LIN {X 0,Y 580.276,Z 358.823,A -85,B 0,C 180,E1 -1965.982,E2 -1965.982} C_VEL
LIN {X 0,Y 580.288,Z 358.825,A -85,B 0,C 180,E1 -1968.827,E2 -1968.827} C_VEL
LIN {X 0,Y 580.269,Z 358.822,A -85,B 0,C 180,E1 -1971.643,E2 -1971.643} C_VEL
LIN {X 0,Y 580.294,Z 358.829,A -85,B 0,C 180,E1 -1974.44,E2 -1974.44} C_VEL
LIN {X 0,Y 580.294,Z 358.821,A -85,B 0,C 180,E1 -1977.223,E2 -1977.223} C_VEL
LIN {X 0,Y 580.311,Z 358.82,A -85,B 0,C 180,E1 -1980,E2 -1980} C_VEL
LIN {X 0,Y 580.319,Z 358.824,A -85,B 0,C 180,E1 -1982.777,E2 -1982.777} C_VEL
LIN {X 0,Y 580.273,Z 358.822,A -85,B 0,C 180,E1 -1985.56,E2 -1985.56} C_VEL
LIN {X 0,Y 580.238,Z 358.826,A -85,B 0,C 180,E1 -1987.657,E2 -1987.657} C_VEL
LIN {X 0,Y 580.25,Z 358.833,A -85,B 0,C 180,E1 -1990.468,E2 -1990.468} C_VEL
LIN {X 0,Y 580.275,Z 358.83,A -85,B 0,C 180,E1 -1992.592,E2 -1992.592} C_VEL
LIN {X 0,Y 580.261,Z 358.824,A -85,B 0,C 180,E1 -1995.454,E2 -1995.454} C_VEL
LIN {X 0,Y 580.245,Z 358.825,A -85,B 0,C 180,E1 -1997.626,E2 -1997.626} C_VEL
LIN {X 0,Y 580.26,Z 358.824,A -85,B 0,C 180,E1 -1999.824,E2 -1999.824} C_VEL
LIN {X 0,Y 580.262,Z 358.824,A -85,B 0,C 180,E1 -2001.343,E2 -2001.343} C_VEL
LIN {X 0,Y 579.556,Z 358.913,A -85,B 0,C 180,E1 -2001.923,E2 -2001.923} C_VEL
LIN {X 0,Y 576.673,Z 359.279,A -85,B 0,C 180,E1 -2002.862,E2 -2002.862} C_VEL
LIN {X 0,Y 574.271,Z 359.574,A -85,B 0,C 180,E1 -2003.618,E2 -2003.618} C_VEL
LIN {X 0,Y 573.259,Z 359.7,A -85,B 0,C 180,E1 -2004.202,E2 -2004.202} C_VEL
LIN {X 0,Y 573.185,Z 359.711,A -85,B 0,C 180,E1 -2004.4,E2 -2004.4} C_VEL
LIN {X 0,Y 573.168,Z 359.714,A -85,B 0,C 180,E1 -2006.98,E2 -2006.98} C_VEL
LIN {X 0,Y 573.197,Z 359.704,A -85,B 0,C 180,E1 -2009.483,E2 -2009.483} C_VEL
LIN {X 0,Y 573.224,Z 359.704,A -85,B 0,C 180,E1 -2012.227,E2 -2012.227} C_VEL
LIN {X 0,Y 573.213,Z 359.712,A -85,B 0,C 180,E1 -2014.771,E2 -2014.771} C_VEL
LIN {X 0,Y 573.201,Z 359.7,A -85,B 0,C 180,E1 -2017.81,E2 -2017.81} C_VEL
LIN {X 0,Y 573.233,Z 359.706,A -85,B 0,C 180,E1 -2020.526,E2 -2020.526} C_VEL
LIN {X 0,Y 573.191,Z 359.705,A -85,B 0,C 180,E1 -2023.666,E2 -2023.666} C_VEL
LIN {X 0,Y 573.184,Z 359.713,A -85,B 0,C 180,E1 -2026.638,E2 -2026.638} C_VEL
LIN {X 0,Y 573.218,Z 359.702,A -85,B 0,C 180,E1 -2029.478,E2 -2029.478} C_VEL
LIN {X 0,Y 573.21,Z 359.705,A -85,B 0,C 180,E1 -2032.192,E2 -2032.192} C_VEL
LIN {X 0,Y 573.205,Z 359.703,A -85,B 0,C 180,E1 -2035.233,E2 -2035.233} C_VEL
LIN {X 0,Y 573.226,Z 359.706,A -85,B 0,C 180,E1 -2037.776,E2 -2037.776} C_VEL
LIN {X 0,Y 573.237,Z 359.888,A -85,B 0,C 180,E1 -2039.418,E2 -2039.418} C_VEL
LIN {X 0,Y 575.578,Z 368.52,A -85,B 0,C 180,E1 -2040.393,E2 -2040.393} C_VEL
LIN {X 0,Y 575.413,Z 394.138,A -85,B 0,C 180,E1 -2042.851,E2 -2042.851} C_VEL
LIN {X 0,Y 574.972,Z 420.796,A -85,B 0,C 180,E1 -2045.445,E2 -2045.445} C_VEL
LIN {X 0,Y 574.579,Z 450.721,A -85,B 0,C 180,E1 -2048.305,E2 -2048.305} C_VEL
LIN {X 0,Y 574.313,Z 473.19,A -85,B 0,C 180,E1 -2050.401,E2 -2050.401} C_VEL
LIN {X 0,Y 575.197,Z 479.4,A -85,B 0,C 180,E1 -2050.536,E2 -2050.536} C_VEL
LIN {X 0,Y 574.747,Z 640.976,A -85,B 0,C 180,E1 -2052.626,E2 -2052.626} C_VEL
LIN {X 0,Y 574.62,Z 656.727,A -85,B 0,C 180,E1 -2052.977,E2 -2052.977} C_VEL
LIN {X 0,Y 574.428,Z 672.064,A -85,B 0,C 180,E1 -2053.475,E2 -2053.475} C_VEL
LIN {X 0,Y 574.244,Z 686.728,A -85,B 0,C 180,E1 -2054.108,E2 -2054.108} C_VEL
LIN {X 0,Y 574.017,Z 700.024,A -85,B 0,C 180,E1 -2054.83,E2 -2054.83} C_VEL
LIN {X 0,Y 573.856,Z 713.545,A -85,B 0,C 180,E1 -2055.73,E2 -2055.73} C_VEL
LIN {X 0,Y 573.629,Z 725.875,A -85,B 0,C 180,E1 -2056.721,E2 -2056.721} C_VEL
LIN {X 0,Y 573.455,Z 737.075,A -85,B 0,C 180,E1 -2057.796,E2 -2057.796} C_VEL
LIN {X 0,Y 573.294,Z 746.586,A -85,B 0,C 180,E1 -2058.877,E2 -2058.877} C_VEL
LIN {X 0,Y 573.202,Z 755.792,A -85,B 0,C 180,E1 -2060.117,E2 -2060.117} C_VEL
LIN {X 0,Y 573.133,Z 763.502,A -85,B 0,C 180,E1 -2061.362,E2 -2061.362} C_VEL
LIN {X 0,Y 573.074,Z 769.895,A -85,B 0,C 180,E1 -2062.603,E2 -2062.603} C_VEL
LIN {X 0,Y 573.04,Z 775.776,A -85,B 0,C 180,E1 -2064.017,E2 -2064.017} C_VEL
LIN {X 0,Y 572.949,Z 779.256,A -85,B 0,C 180,E1 -2065.075,E2 -2065.075} C_VEL
LIN {X 0,Y 573.004,Z 782.795,A -85,B 0,C 180,E1 -2066.485,E2 -2066.485} C_VEL
LIN {X 0,Y 572.938,Z 785.142,A -85,B 0,C 180,E1 -2067.892,E2 -2067.892} C_VEL
LIN {X 0,Y 572.936,Z 786.338,A -85,B 0,C 180,E1 -2069.298,E2 -2069.298} C_VEL
LIN {X 0,Y 572.937,Z 786.36,A -85,B 0,C 180,E1 -2070.704,E2 -2070.704} C_VEL
LIN {X 0,Y 572.938,Z 785.241,A -85,B 0,C 180,E1 -2072.11,E2 -2072.11} C_VEL
LIN {X 0,Y 573.006,Z 782.976,A -85,B 0,C 180,E1 -2073.517,E2 -2073.517} C_VEL
LIN {X 0,Y 572.95,Z 779.516,A -85,B 0,C 180,E1 -2074.927,E2 -2074.927} C_VEL
LIN {X 0,Y 573.008,Z 774.781,A -85,B 0,C 180,E1 -2076.339,E2 -2076.339} C_VEL
LIN {X 0,Y 573.085,Z 768.641,A -85,B 0,C 180,E1 -2077.754,E2 -2077.754} C_VEL
LIN {X 0,Y 573.134,Z 760.919,A -85,B 0,C 180,E1 -2079.174,E2 -2079.174} C_VEL
LIN {X 0,Y 573.266,Z 752.685,A -85,B 0,C 180,E1 -2080.419,E2 -2080.419} C_VEL
LIN {X 0,Y 573.358,Z 742.768,A -85,B 0,C 180,E1 -2081.67,E2 -2081.67} C_VEL
LIN {X 0,Y 573.535,Z 732.642,A -85,B 0,C 180,E1 -2082.743,E2 -2082.743} C_VEL
LIN {X 0,Y 573.723,Z 720.552,A -85,B 0,C 180,E1 -2083.821,E2 -2083.821} C_VEL
LIN {X 0,Y 573.921,Z 707.579,A -85,B 0,C 180,E1 -2084.781,E2 -2084.781} C_VEL
LIN {X 0,Y 574.108,Z 693.671,A -85,B 0,C 180,E1 -2085.624,E2 -2085.624} C_VEL
LIN {X 0,Y 574.347,Z 678.714,A -85,B 0,C 180,E1 -2086.347,E2 -2086.347} C_VEL
LIN {X 0,Y 574.522,Z 664.182,A -85,B 0,C 180,E1 -2086.891,E2 -2086.891} C_VEL
LIN {X 0,Y 574.678,Z 648.349,A -85,B 0,C 180,E1 -2087.319,E2 -2087.319} C_VEL
LIN {X 0,Y 574.802,Z 632.324,A -85,B 0,C 180,E1 -2087.594,E2 -2087.594} C_VEL
LIN {X 0,Y 575.072,Z 478.201,A -85,B 0,C 180,E1 -2089.574,E2 -2089.574} C_VEL
LIN {X 0,Y 574.313,Z 473.126,A -85,B 0,C 180,E1 -2089.693,E2 -2089.693} C_VEL
LIN {X 0,Y 574.658,Z 443.511,A -85,B 0,C 180,E1 -2092.47,E2 -2092.47} C_VEL
LIN {X 0,Y 575.119,Z 413.767,A -85,B 0,C 180,E1 -2095.323,E2 -2095.323} C_VEL
LIN {X 0,Y 575.538,Z 385.83,A -85,B 0,C 180,E1 -2098.033,E2 -2098.033} C_VEL
LIN {X 0,Y 575.647,Z 369.112,A -85,B 0,C 180,E1 -2099.635,E2 -2099.635} C_VEL
LIN {X 0,Y 573.219,Z 359.876,A -85,B 0,C 180,E1 -2100.676,E2 -2100.676} C_VEL
LIN {X 0,Y 573.181,Z 359.705,A -85,B 0,C 180,E1 -2103.511,E2 -2103.511} C_VEL
LIN {X 0,Y 573.177,Z 359.708,A -85,B 0,C 180,E1 -2106.055,E2 -2106.055} C_VEL
LIN {X 0,Y 573.175,Z 359.711,A -85,B 0,C 180,E1 -2108.708,E2 -2108.708} C_VEL
LIN {X 0,Y 573.187,Z 359.707,A -85,B 0,C 180,E1 -2111.588,E2 -2111.588} C_VEL
LIN {X 0,Y 573.204,Z 359.704,A -85,B 0,C 180,E1 -2114.337,E2 -2114.337} C_VEL
LIN {X 0,Y 573.208,Z 359.71,A -85,B 0,C 180,E1 -2117.363,E2 -2117.363} C_VEL
LIN {X 0,Y 573.23,Z 359.698,A -85,B 0,C 180,E1 -2120.571,E2 -2120.571} C_VEL
LIN {X 0,Y 573.222,Z 359.711,A -85,B 0,C 180,E1 -2123.075,E2 -2123.075} C_VEL
LIN {X 0,Y 573.241,Z 359.699,A -85,B 0,C 180,E1 -2125.669,E2 -2125.669} C_VEL
LIN {X 0,Y 573.222,Z 359.702,A -85,B 0,C 180,E1 -2128.183,E2 -2128.183} C_VEL
LIN {X 0,Y 573.229,Z 359.703,A -85,B 0,C 180,E1 -2130.632,E2 -2130.632} C_VEL
LIN {X 0,Y 573.196,Z 359.709,A -85,B 0,C 180,E1 -2133.517,E2 -2133.517} C_VEL
LIN {X 0,Y 573.2,Z 359.705,A -85,B 0,C 180,E1 -2136.133,E2 -2136.133} C_VEL
LIN {X 0,Y 573.25,Z 359.707,A -85,B 0,C 180,E1 -2139.174,E2 -2139.174} C_VEL
LIN {X 0,Y 573.266,Z 359.908,A -85,B 0,C 180,E1 -2140.67,E2 -2140.67} C_VEL
LIN {X 0,Y 573.579,Z 364.187,A -85,B 0,C 180,E1 -2141.423,E2 -2141.423} C_VEL
LIN {X 0,Y 573.483,Z 375.119,A -85,B 0,C 180,E1 -2143.226,E2 -2143.226} C_VEL
LIN {X 0,Y 573.795,Z 377.158,A -85,B 0,C 180,E1 -2143.334,E2 -2143.334} C_VEL
LIN {X 0,Y 574.525,Z 380.871,A -85,B 0,C 180,E1 -2143.403,E2 -2143.403} C_VEL
LIN {X 0,Y 574.282,Z 511.941,A -85,B 0,C 180,E1 -2145.085,E2 -2145.085} C_VEL
LIN {X 0,Y 574.209,Z 526.01,A -85,B 0,C 180,E1 -2145.412,E2 -2145.412} C_VEL
LIN {X 0,Y 574.033,Z 539.748,A -85,B 0,C 180,E1 -2145.871,E2 -2145.871} C_VEL
LIN {X 0,Y 573.895,Z 552.81,A -85,B 0,C 180,E1 -2146.455,E2 -2146.455} C_VEL
LIN {X 0,Y 573.722,Z 565.419,A -85,B 0,C 180,E1 -2147.172,E2 -2147.172} C_VEL
LIN {X 0,Y 573.531,Z 578.049,A -85,B 0,C 180,E1 -2148.066,E2 -2148.066} C_VEL
LIN {X 0,Y 573.439,Z 589.713,A -85,B 0,C 180,E1 -2149.082,E2 -2149.082} C_VEL
LIN {X 0,Y 573.236,Z 599.474,A -85,B 0,C 180,E1 -2150.117,E2 -2150.117} C_VEL
LIN {X 0,Y 573.203,Z 607.851,A -85,B 0,C 180,E1 -2151.184,E2 -2151.184} C_VEL
LIN {X 0,Y 573.112,Z 615.879,A -85,B 0,C 180,E1 -2152.425,E2 -2152.425} C_VEL
LIN {X 0,Y 573.021,Z 622.341,A -85,B 0,C 180,E1 -2153.663,E2 -2153.663} C_VEL
LIN {X 0,Y 573.001,Z 626.782,A -85,B 0,C 180,E1 -2154.722,E2 -2154.722} C_VEL
LIN {X 0,Y 573.028,Z 630.325,A -85,B 0,C 180,E1 -2155.78,E2 -2155.78} C_VEL
LIN {X 0,Y 572.957,Z 633.74,A -85,B 0,C 180,E1 -2157.188,E2 -2157.188} C_VEL
LIN {X 0,Y 572.944,Z 635.776,A -85,B 0,C 180,E1 -2158.594,E2 -2158.594} C_VEL
LIN {X 0,Y 572.935,Z 636.496,A -85,B 0,C 180,E1 -2160,E2 -2160} C_VEL
LIN {X 0,Y 572.941,Z 635.879,A -85,B 0,C 180,E1 -2161.406,E2 -2161.406} C_VEL
LIN {X 0,Y 572.957,Z 633.92,A -85,B 0,C 180,E1 -2162.812,E2 -2162.812} C_VEL
LIN {X 0,Y 573.03,Z 630.578,A -85,B 0,C 180,E1 -2164.22,E2 -2164.22} C_VEL
LIN {X 0,Y 573.056,Z 625.765,A -85,B 0,C 180,E1 -2165.63,E2 -2165.63} C_VEL
LIN {X 0,Y 573.055,Z 619.303,A -85,B 0,C 180,E1 -2167.044,E2 -2167.044} C_VEL
LIN {X 0,Y 573.143,Z 612.104,A -85,B 0,C 180,E1 -2168.284,E2 -2168.284} C_VEL
LIN {X 0,Y 573.226,Z 603.16,A -85,B 0,C 180,E1 -2169.527,E2 -2169.527} C_VEL
LIN {X 0,Y 573.351,Z 593.818,A -85,B 0,C 180,E1 -2170.595,E2 -2170.595} C_VEL
LIN {X 0,Y 573.469,Z 583.594,A -85,B 0,C 180,E1 -2171.567,E2 -2171.567} C_VEL
LIN {X 0,Y 573.627,Z 572.102,A -85,B 0,C 180,E1 -2172.471,E2 -2172.471} C_VEL
LIN {X 0,Y 573.77,Z 559.465,A -85,B 0,C 180,E1 -2173.277,E2 -2173.277} C_VEL
LIN {X 0,Y 573.992,Z 546.16,A -85,B 0,C 180,E1 -2173.949,E2 -2173.949} C_VEL
LIN {X 0,Y 574.133,Z 531.721,A -85,B 0,C 180,E1 -2174.506,E2 -2174.506} C_VEL
LIN {X 0,Y 574.237,Z 517.562,A -85,B 0,C 180,E1 -2174.893,E2 -2174.893} C_VEL
LIN {X 0,Y 574.296,Z 502.798,A -85,B 0,C 180,E1 -2175.141,E2 -2175.141} C_VEL
LIN {X 0,Y 574.492,Z 380.765,A -85,B 0,C 180,E1 -2176.689,E2 -2176.689} C_VEL
LIN {X 0,Y 573.474,Z 375.534,A -85,B 0,C 180,E1 -2176.814,E2 -2176.814} C_VEL
LIN {X 0,Y 573.534,Z 368.013,A -85,B 0,C 180,E1 -2178.024,E2 -2178.024} C_VEL
LIN {X 0,Y 573.603,Z 362.527,A -85,B 0,C 180,E1 -2178.947,E2 -2178.947} C_VEL
LIN {X 0,Y 573.257,Z 359.762,A -85,B 0,C 180,E1 -2179.516,E2 -2179.516} C_VEL
LIN {X 0,Y 573.235,Z 359.706,A -85,B 0,C 180,E1 -2182.338,E2 -2182.338} C_VEL
LIN {X 0,Y 573.258,Z 359.7,A -85,B 0,C 180,E1 -2185.41,E2 -2185.41} C_VEL
LIN {X 0,Y 573.25,Z 359.7,A -85,B 0,C 180,E1 -2188.028,E2 -2188.028} C_VEL
LIN {X 0,Y 573.249,Z 359.702,A -85,B 0,C 180,E1 -2190.176,E2 -2190.176} C_VEL
LIN {X 0,Y 573.257,Z 359.707,A -85,B 0,C 180,E1 -2192.645,E2 -2192.645} C_VEL
LIN {X 0,Y 573.211,Z 359.705,A -85,B 0,C 180,E1 -2195.188,E2 -2195.188} C_VEL
LIN {X 0,Y 573.233,Z 359.703,A -85,B 0,C 180,E1 -2197.808,E2 -2197.808} C_VEL
LIN {X 0,Y 573.249,Z 359.706,A -85,B 0,C 180,E1 -2200.525,E2 -2200.525} C_VEL
LIN {X 0,Y 573.211,Z 359.704,A -85,B 0,C 180,E1 -2203.362,E2 -2203.362} C_VEL
LIN {X 0,Y 573.209,Z 359.712,A -85,B 0,C 180,E1 -2206.335,E2 -2206.335} C_VEL
LIN {X 0,Y 573.207,Z 359.709,A -85,B 0,C 180,E1 -2208.54,E2 -2208.54} C_VEL
LIN {X 0,Y 573.232,Z 359.702,A -85,B 0,C 180,E1 -2211.297,E2 -2211.297} C_VEL
LIN {X 0,Y 573.184,Z 359.716,A -85,B 0,C 180,E1 -2214.022,E2 -2214.022} C_VEL
LIN {X 0,Y 573.224,Z 359.706,A -85,B 0,C 180,E1 -2216.514,E2 -2216.514} C_VEL
LIN {X 0,Y 573.208,Z 359.709,A -85,B 0,C 180,E1 -2219.121,E2 -2219.121} C_VEL
LIN {X 0,Y 573.247,Z 359.929,A -85,B 0,C 180,E1 -2220.32,E2 -2220.32} C_VEL
LIN {X 0,Y 575.631,Z 368.055,A -85,B 0,C 180,E1 -2221.166,E2 -2221.166} C_VEL
LIN {X 0,Y 575.545,Z 389.554,A -85,B 0,C 180,E1 -2223.05,E2 -2223.05} C_VEL
LIN {X 0,Y 575.1,Z 418.496,A -85,B 0,C 180,E1 -2225.641,E2 -2225.641} C_VEL
LIN {X 0,Y 574.621,Z 451.836,A -85,B 0,C 180,E1 -2228.567,E2 -2228.567} C_VEL
LIN {X 0,Y 574.433,Z 472.925,A -85,B 0,C 180,E1 -2230.37,E2 -2230.37} C_VEL
LIN {X 0,Y 575.2,Z 478.523,A -85,B 0,C 180,E1 -2230.48,E2 -2230.48} C_VEL
LIN {X 0,Y 574.764,Z 641.003,A -85,B 0,C 180,E1 -2232.58,E2 -2232.58} C_VEL
LIN {X 0,Y 574.631,Z 656.684,A -85,B 0,C 180,E1 -2232.93,E2 -2232.93} C_VEL
LIN {X 0,Y 574.413,Z 672.024,A -85,B 0,C 180,E1 -2233.426,E2 -2233.426} C_VEL
LIN {X 0,Y 574.293,Z 685.745,A -85,B 0,C 180,E1 -2234.016,E2 -2234.016} C_VEL
LIN {X 0,Y 574.05,Z 699.226,A -85,B 0,C 180,E1 -2234.738,E2 -2234.738} C_VEL
LIN {X 0,Y 573.863,Z 712.808,A -85,B 0,C 180,E1 -2235.631,E2 -2235.631} C_VEL
LIN {X 0,Y 573.636,Z 725.34,A -85,B 0,C 180,E1 -2236.628,E2 -2236.628} C_VEL
LIN {X 0,Y 573.478,Z 735.739,A -85,B 0,C 180,E1 -2237.615,E2 -2237.615} C_VEL
LIN {X 0,Y 573.288,Z 745.763,A -85,B 0,C 180,E1 -2238.733,E2 -2238.733} C_VEL
LIN {X 0,Y 573.243,Z 754.85,A -85,B 0,C 180,E1 -2239.937,E2 -2239.937} C_VEL
LIN {X 0,Y 573.133,Z 762.724,A -85,B 0,C 180,E1 -2241.182,E2 -2241.182} C_VEL
LIN {X 0,Y 573.076,Z 770.083,A -85,B 0,C 180,E1 -2242.601,E2 -2242.601} C_VEL
LIN {X 0,Y 573.04,Z 775.921,A -85,B 0,C 180,E1 -2244.015,E2 -2244.015} C_VEL
LIN {X 0,Y 572.951,Z 779.382,A -85,B 0,C 180,E1 -2245.073,E2 -2245.073} C_VEL
LIN {X 0,Y 573.005,Z 782.885,A -85,B 0,C 180,E1 -2246.483,E2 -2246.483} C_VEL
LIN {X 0,Y 572.935,Z 785.19,A -85,B 0,C 180,E1 -2247.89,E2 -2247.89} C_VEL
LIN {X 0,Y 572.938,Z 786.349,A -85,B 0,C 180,E1 -2249.296,E2 -2249.296} C_VEL
LIN {X 0,Y 572.938,Z 786.35,A -85,B 0,C 180,E1 -2250.702,E2 -2250.702} C_VEL
LIN {X 0,Y 572.935,Z 785.194,A -85,B 0,C 180,E1 -2252.108,E2 -2252.108} C_VEL
LIN {X 0,Y 573.004,Z 782.891,A -85,B 0,C 180,E1 -2253.515,E2 -2253.515} C_VEL
LIN {X 0,Y 572.951,Z 779.388,A -85,B 0,C 180,E1 -2254.925,E2 -2254.925} C_VEL
LIN {X 0,Y 573.011,Z 774.611,A -85,B 0,C 180,E1 -2256.336,E2 -2256.336} C_VEL
LIN {X 0,Y 573.095,Z 768.431,A -85,B 0,C 180,E1 -2257.751,E2 -2257.751} C_VEL
LIN {X 0,Y 573.14,Z 760.659,A -85,B 0,C 180,E1 -2259.171,E2 -2259.171} C_VEL
LIN {X 0,Y 573.269,Z 752.378,A -85,B 0,C 180,E1 -2260.417,E2 -2260.417} C_VEL
LIN {X 0,Y 573.384,Z 742.402,A -85,B 0,C 180,E1 -2261.667,E2 -2261.667} C_VEL
LIN {X 0,Y 573.566,Z 732.202,A -85,B 0,C 180,E1 -2262.74,E2 -2262.74} C_VEL
LIN {X 0,Y 573.742,Z 720.03,A -85,B 0,C 180,E1 -2263.818,E2 -2263.818} C_VEL
LIN {X 0,Y 573.958,Z 706.919,A -85,B 0,C 180,E1 -2264.78,E2 -2264.78} C_VEL
LIN {X 0,Y 574.109,Z 694.544,A -85,B 0,C 180,E1 -2265.531,E2 -2265.531} C_VEL
LIN {X 0,Y 574.352,Z 679.863,A -85,B 0,C 180,E1 -2266.253,E2 -2266.253} C_VEL
LIN {X 0,Y 574.544,Z 665.646,A -85,B 0,C 180,E1 -2266.796,E2 -2266.796} C_VEL
LIN {X 0,Y 574.661,Z 650.585,A -85,B 0,C 180,E1 -2267.223,E2 -2267.223} C_VEL
LIN {X 0,Y 574.756,Z 635.683,A -85,B 0,C 180,E1 -2267.502,E2 -2267.502} C_VEL
LIN {X 0,Y 575.134,Z 477.69,A -85,B 0,C 180,E1 -2269.534,E2 -2269.534} C_VEL
LIN {X 0,Y 574.392,Z 472.458,A -85,B 0,C 180,E1 -2269.657,E2 -2269.657} C_VEL
LIN {X 0,Y 574.814,Z 438.957,A -85,B 0,C 180,E1 -2272.556,E2 -2272.556} C_VEL
LIN {X 0,Y 575.287,Z 405.617,A -85,B 0,C 180,E1 -2275.506,E2 -2275.506} C_VEL
LIN {X 0,Y 575.728,Z 377.32,A -85,B 0,C 180,E1 -2278.031,E2 -2278.031} C_VEL
LIN {X 0,Y 575.712,Z 368.417,A -85,B 0,C 180,E1 -2278.827,E2 -2278.827} C_VEL
LIN {X 0,Y 573.241,Z 359.903,A -85,B 0,C 180,E1 -2279.75,E2 -2279.75} C_VEL
LIN {X 0,Y 573.235,Z 359.706,A -85,B 0,C 180,E1 -2282.644,E2 -2282.644} C_VEL
LIN {X 0,Y 573.173,Z 359.708,A -85,B 0,C 180,E1 -2285.188,E2 -2285.188} C_VEL
LIN {X 0,Y 573.206,Z 359.707,A -85,B 0,C 180,E1 -2287.808,E2 -2287.808} C_VEL
LIN {X 0,Y 573.234,Z 359.707,A -85,B 0,C 180,E1 -2290.524,E2 -2290.524} C_VEL
LIN {X 0,Y 573.193,Z 359.705,A -85,B 0,C 180,E1 -2293.361,E2 -2293.361} C_VEL
LIN {X 0,Y 573.182,Z 359.713,A -85,B 0,C 180,E1 -2296.335,E2 -2296.335} C_VEL
LIN {X 0,Y 573.232,Z 359.698,A -85,B 0,C 180,E1 -2299.474,E2 -2299.474} C_VEL
LIN {X 0,Y 573.2,Z 359.711,A -85,B 0,C 180,E1 -2302.19,E2 -2302.19} C_VEL
LIN {X 0,Y 573.206,Z 359.698,A -85,B 0,C 180,E1 -2305.23,E2 -2305.23} C_VEL
LIN {X 0,Y 573.221,Z 359.702,A -85,B 0,C 180,E1 -2307.774,E2 -2307.774} C_VEL
LIN {X 0,Y 573.223,Z 359.707,A -85,B 0,C 180,E1 -2310.632,E2 -2310.632} C_VEL
LIN {X 0,Y 573.192,Z 359.705,A -85,B 0,C 180,E1 -2313.513,E2 -2313.513} C_VEL
LIN {X 0,Y 573.183,Z 359.709,A -85,B 0,C 180,E1 -2316.132,E2 -2316.132} C_VEL
LIN {X 0,Y 573.218,Z 359.706,A -85,B 0,C 180,E1 -2318.713,E2 -2318.713} C_VEL
LIN {X 0,Y 573.178,Z 359.706,A -85,B 0,C 180,E1 -2321.41,E2 -2321.41} C_VEL
LIN {X 0,Y 573.19,Z 359.713,A -85,B 0,C 180,E1 -2324.351,E2 -2324.351} C_VEL
LIN {X 0,Y 573.182,Z 359.715,A -85,B 0,C 180,E1 -2326.528,E2 -2326.528} C_VEL
LIN {X 0,Y 573.219,Z 359.7,A -85,B 0,C 180,E1 -2329.403,E2 -2329.403} C_VEL
LIN {X 0,Y 573.219,Z 359.706,A -85,B 0,C 180,E1 -2332.249,E2 -2332.249} C_VEL
LIN {X 0,Y 573.263,Z 359.696,A -85,B 0,C 180,E1 -2335.077,E2 -2335.077} C_VEL
LIN {X 0,Y 573.269,Z 359.696,A -85,B 0,C 180,E1 -2337.892,E2 -2337.892} C_VEL
LIN {X 0,Y 573.316,Z 359.695,A -85,B 0,C 180,E1 -2340.702,E2 -2340.702} C_VEL
LIN {X 0,Y 573.282,Z 359.7,A -85,B 0,C 180,E1 -2342.811,E2 -2342.811} C_VEL
LIN {X 0,Y 573.242,Z 359.697,A -85,B 0,C 180,E1 -2345.629,E2 -2345.629} C_VEL
LIN {X 0,Y 573.196,Z 359.703,A -85,B 0,C 180,E1 -2347.751,E2 -2347.751} C_VEL
LIN {X 0,Y 573.225,Z 359.71,A -85,B 0,C 180,E1 -2350.597,E2 -2350.597} C_VEL
LIN {X 0,Y 573.194,Z 359.704,A -85,B 0,C 180,E1 -2353.472,E2 -2353.472} C_VEL
LIN {X 0,Y 573.203,Z 359.702,A -85,B 0,C 180,E1 -2355.649,E2 -2355.649} C_VEL
LIN {X 0,Y 573.204,Z 359.703,A -85,B 0,C 180,E1 -2357.85,E2 -2357.85} C_VEL
LIN {X 0,Y 573.218,Z 359.703,A -85,B 0,C 180,E1 -2360.078,E2 -2360.078} C_VEL
LIN {X 0,Y 573.204,Z 359.707,A -85,B 0,C 180,E1 -2362.339,E2 -2362.339} C_VEL
LIN {X 0,Y 573.185,Z 359.711,A -85,B 0,C 180,E1 -2364.4,E2 -2364.4} C_VEL
LIN {X 0,Y 572.543,Z 359.797,A -85,B 0,C 180,E1 -2364.986,E2 -2364.986} C_VEL
LIN {X 0,Y 569.696,Z 360.152,A -85,B 0,C 180,E1 -2365.938,E2 -2365.938} C_VEL
LIN {X 0,Y 567.272,Z 360.451,A -85,B 0,C 180,E1 -2366.703,E2 -2366.703} C_VEL
LIN {X 0,Y 566.225,Z 360.575,A -85,B 0,C 180,E1 -2367.295,E2 -2367.295} C_VEL
LIN {X 0,Y 566.138,Z 360.584,A -85,B 0,C 180,E1 -2367.495,E2 -2367.495} C_VEL
LIN {X 0,Y 566.144,Z 360.582,A -85,B 0,C 180,E1 -2369.772,E2 -2369.772} C_VEL
LIN {X 0,Y 566.178,Z 360.584,A -85,B 0,C 180,E1 -2372.429,E2 -2372.429} C_VEL
LIN {X 0,Y 566.157,Z 360.587,A -85,B 0,C 180,E1 -2374.989,E2 -2374.989} C_VEL
LIN {X 0,Y 566.17,Z 360.576,A -85,B 0,C 180,E1 -2377.463,E2 -2377.463} C_VEL
LIN {X 0,Y 566.191,Z 360.579,A -85,B 0,C 180,E1 -2380.201,E2 -2380.201} C_VEL
LIN {X 0,Y 566.164,Z 360.586,A -85,B 0,C 180,E1 -2383.058,E2 -2383.058} C_VEL
LIN {X 0,Y 566.135,Z 360.584,A -85,B 0,C 180,E1 -2386.056,E2 -2386.056} C_VEL
LIN {X 0,Y 566.151,Z 360.585,A -85,B 0,C 180,E1 -2389.221,E2 -2389.221} C_VEL
LIN {X 0,Y 566.161,Z 360.583,A -85,B 0,C 180,E1 -2391.637,E2 -2391.637} C_VEL
LIN {X 0,Y 566.122,Z 360.59,A -85,B 0,C 180,E1 -2394.307,E2 -2394.307} C_VEL
LIN {X 0,Y 566.155,Z 360.576,A -85,B 0,C 180,E1 -2396.895,E2 -2396.895} C_VEL
LIN {X 0,Y 566.188,Z 360.808,A -85,B 0,C 180,E1 -2399.168,E2 -2399.168} C_VEL
LIN {X 0,Y 568.738,Z 369.93,A -85,B 0,C 180,E1 -2400.206,E2 -2400.206} C_VEL
LIN {X 0,Y 568.844,Z 380.062,A -85,B 0,C 180,E1 -2401.196,E2 -2401.196} C_VEL
LIN {X 0,Y 568.492,Z 410.872,A -85,B 0,C 180,E1 -2404.167,E2 -2404.167} C_VEL
LIN {X 0,Y 567.948,Z 440.619,A -85,B 0,C 180,E1 -2407.06,E2 -2407.06} C_VEL
LIN {X 0,Y 567.49,Z 470.21,A -85,B 0,C 180,E1 -2409.888,E2 -2409.888} C_VEL
LIN {X 0,Y 567.499,Z 473.493,A -85,B 0,C 180,E1 -2410.169,E2 -2410.169} C_VEL
LIN {X 0,Y 568.505,Z 481.039,A -85,B 0,C 180,E1 -2410.318,E2 -2410.318} C_VEL
LIN {X 0,Y 567.992,Z 640.989,A -85,B 0,C 180,E1 -2412.412,E2 -2412.412} C_VEL
LIN {X 0,Y 567.869,Z 655.887,A -85,B 0,C 180,E1 -2412.746,E2 -2412.746} C_VEL
LIN {X 0,Y 567.629,Z 670.839,A -85,B 0,C 180,E1 -2413.225,E2 -2413.225} C_VEL
LIN {X 0,Y 567.412,Z 684.828,A -85,B 0,C 180,E1 -2413.82,E2 -2413.82} C_VEL
LIN {X 0,Y 567.173,Z 698.498,A -85,B 0,C 180,E1 -2414.55,E2 -2414.55} C_VEL
LIN {X 0,Y 566.955,Z 711.028,A -85,B 0,C 180,E1 -2415.368,E2 -2415.368} C_VEL
LIN {X 0,Y 566.676,Z 723.792,A -85,B 0,C 180,E1 -2416.372,E2 -2416.372} C_VEL
LIN {X 0,Y 566.504,Z 735.333,A -85,B 0,C 180,E1 -2417.462,E2 -2417.462} C_VEL
LIN {X 0,Y 566.348,Z 745.626,A -85,B 0,C 180,E1 -2418.62,E2 -2418.62} C_VEL
LIN {X 0,Y 566.22,Z 754.57,A -85,B 0,C 180,E1 -2419.814,E2 -2419.814} C_VEL
LIN {X 0,Y 566.077,Z 763.507,A -85,B 0,C 180,E1 -2421.253,E2 -2421.253} C_VEL
LIN {X 0,Y 565.997,Z 769.899,A -85,B 0,C 180,E1 -2422.51,E2 -2422.51} C_VEL
LIN {X 0,Y 565.957,Z 775.779,A -85,B 0,C 180,E1 -2423.942,E2 -2423.942} C_VEL
LIN {X 0,Y 565.865,Z 779.257,A -85,B 0,C 180,E1 -2425.014,E2 -2425.014} C_VEL
LIN {X 0,Y 565.909,Z 782.797,A -85,B 0,C 180,E1 -2426.441,E2 -2426.441} C_VEL
LIN {X 0,Y 565.838,Z 785.142,A -85,B 0,C 180,E1 -2427.866,E2 -2427.866} C_VEL
LIN {X 0,Y 565.836,Z 786.338,A -85,B 0,C 180,E1 -2429.289,E2 -2429.289} C_VEL
LIN {X 0,Y 565.837,Z 786.36,A -85,B 0,C 180,E1 -2430.713,E2 -2430.713} C_VEL
LIN {X 0,Y 565.839,Z 785.241,A -85,B 0,C 180,E1 -2432.136,E2 -2432.136} C_VEL
LIN {X 0,Y 565.911,Z 782.975,A -85,B 0,C 180,E1 -2433.561,E2 -2433.561} C_VEL
LIN {X 0,Y 565.865,Z 779.514,A -85,B 0,C 180,E1 -2434.989,E2 -2434.989} C_VEL
LIN {X 0,Y 565.916,Z 774.777,A -85,B 0,C 180,E1 -2436.418,E2 -2436.418} C_VEL
LIN {X 0,Y 566.005,Z 768.637,A -85,B 0,C 180,E1 -2437.851,E2 -2437.851} C_VEL
LIN {X 0,Y 566.068,Z 760.914,A -85,B 0,C 180,E1 -2439.289,E2 -2439.289} C_VEL
LIN {X 0,Y 566.246,Z 752.679,A -85,B 0,C 180,E1 -2440.55,E2 -2440.55} C_VEL
LIN {X 0,Y 566.333,Z 742.76,A -85,B 0,C 180,E1 -2441.816,E2 -2441.816} C_VEL
LIN {X 0,Y 566.553,Z 732.637,A -85,B 0,C 180,E1 -2442.903,E2 -2442.903} C_VEL
LIN {X 0,Y 566.763,Z 720.541,A -85,B 0,C 180,E1 -2443.994,E2 -2443.994} C_VEL
LIN {X 0,Y 566.999,Z 707.976,A -85,B 0,C 180,E1 -2444.938,E2 -2444.938} C_VEL
LIN {X 0,Y 567.225,Z 695.314,A -85,B 0,C 180,E1 -2445.727,E2 -2445.727} C_VEL
LIN {X 0,Y 567.484,Z 680.829,A -85,B 0,C 180,E1 -2446.458,E2 -2446.458} C_VEL
LIN {X 0,Y 567.696,Z 666.907,A -85,B 0,C 180,E1 -2447.007,E2 -2447.007} C_VEL
LIN {X 0,Y 567.876,Z 651.394,A -85,B 0,C 180,E1 -2447.462,E2 -2447.462} C_VEL
LIN {X 0,Y 568.005,Z 635.985,A -85,B 0,C 180,E1 -2447.76,E2 -2447.76} C_VEL
LIN {X 0,Y 568.509,Z 480.221,A -85,B 0,C 180,E1 -2449.782,E2 -2449.782} C_VEL
LIN {X 0,Y 567.5,Z 473.191,A -85,B 0,C 180,E1 -2449.935,E2 -2449.935} C_VEL
LIN {X 0,Y 567.869,Z 443.505,A -85,B 0,C 180,E1 -2452.753,E2 -2452.753} C_VEL
LIN {X 0,Y 568.438,Z 413.76,A -85,B 0,C 180,E1 -2455.642,E2 -2455.642} C_VEL
LIN {X 0,Y 568.779,Z 384.679,A -85,B 0,C 180,E1 -2458.449,E2 -2458.449} C_VEL
LIN {X 0,Y 568.82,Z 370.471,A -85,B 0,C 180,E1 -2459.826,E2 -2459.826} C_VEL
LIN {X 0,Y 566.195,Z 360.766,A -85,B 0,C 180,E1 -2460.935,E2 -2460.935} C_VEL
LIN {X 0,Y 566.145,Z 360.58,A -85,B 0,C 180,E1 -2463.724,E2 -2463.724} C_VEL
LIN {X 0,Y 566.14,Z 360.586,A -85,B 0,C 180,E1 -2466.575,E2 -2466.575} C_VEL
LIN {X 0,Y 566.178,Z 360.583,A -85,B 0,C 180,E1 -2469.681,E2 -2469.681} C_VEL
LIN {X 0,Y 566.148,Z 360.586,A -85,B 0,C 180,E1 -2472.911,E2 -2472.911} C_VEL
LIN {X 0,Y 566.139,Z 360.582,A -85,B 0,C 180,E1 -2475.958,E2 -2475.958} C_VEL
LIN {X 0,Y 566.14,Z 360.589,A -85,B 0,C 180,E1 -2478.857,E2 -2478.857} C_VEL
LIN {X 0,Y 566.181,Z 360.584,A -85,B 0,C 180,E1 -2481.447,E2 -2481.447} C_VEL
LIN {X 0,Y 566.14,Z 360.582,A -85,B 0,C 180,E1 -2484.306,E2 -2484.306} C_VEL
LIN {X 0,Y 566.165,Z 360.583,A -85,B 0,C 180,E1 -2486.894,E2 -2486.894} C_VEL
LIN {X 0,Y 566.161,Z 360.587,A -85,B 0,C 180,E1 -2489.406,E2 -2489.406} C_VEL
LIN {X 0,Y 566.154,Z 360.583,A -85,B 0,C 180,E1 -2491.854,E2 -2491.854} C_VEL
LIN {X 0,Y 566.173,Z 360.58,A -85,B 0,C 180,E1 -2494.249,E2 -2494.249} C_VEL
LIN {X 0,Y 566.164,Z 360.589,A -85,B 0,C 180,E1 -2497.368,E2 -2497.368} C_VEL
LIN {X 0,Y 566.203,Z 360.584,A -85,B 0,C 180,E1 -2499.662,E2 -2499.662} C_VEL
LIN {X 0,Y 566.212,Z 360.704,A -85,B 0,C 180,E1 -2500.492,E2 -2500.492} C_VEL
LIN {X 0,Y 566.619,Z 365.516,A -85,B 0,C 180,E1 -2501.374,E2 -2501.374} C_VEL
LIN {X 0,Y 566.5,Z 372.122,A -85,B 0,C 180,E1 -2502.492,E2 -2502.492} C_VEL
LIN {X 0,Y 566.712,Z 376.347,A -85,B 0,C 180,E1 -2503.036,E2 -2503.036} C_VEL
LIN {X 0,Y 566.99,Z 378.195,A -85,B 0,C 180,E1 -2503.141,E2 -2503.141} C_VEL
LIN {X 0,Y 567.754,Z 382.459,A -85,B 0,C 180,E1 -2503.219,E2 -2503.219} C_VEL
LIN {X 0,Y 567.422,Z 511.965,A -85,B 0,C 180,E1 -2504.901,E2 -2504.901} C_VEL
LIN {X 0,Y 567.334,Z 526.486,A -85,B 0,C 180,E1 -2505.245,E2 -2505.245} C_VEL
LIN {X 0,Y 567.135,Z 540.923,A -85,B 0,C 180,E1 -2505.742,E2 -2505.742} C_VEL
LIN {X 0,Y 566.949,Z 554.548,A -85,B 0,C 180,E1 -2506.377,E2 -2506.377} C_VEL
LIN {X 0,Y 566.746,Z 566.805,A -85,B 0,C 180,E1 -2507.102,E2 -2507.102} C_VEL
LIN {X 0,Y 566.541,Z 579.199,A -85,B 0,C 180,E1 -2508.007,E2 -2508.007} C_VEL
LIN {X 0,Y 566.436,Z 590.057,A -85,B 0,C 180,E1 -2508.979,E2 -2508.979} C_VEL
LIN {X 0,Y 566.209,Z 599.478,A -85,B 0,C 180,E1 -2509.993,E2 -2509.993} C_VEL
LIN {X 0,Y 566.134,Z 607.853,A -85,B 0,C 180,E1 -2511.073,E2 -2511.073} C_VEL
LIN {X 0,Y 566.048,Z 615.88,A -85,B 0,C 180,E1 -2512.33,E2 -2512.33} C_VEL
LIN {X 0,Y 565.947,Z 622.343,A -85,B 0,C 180,E1 -2513.583,E2 -2513.583} C_VEL
LIN {X 0,Y 565.928,Z 626.781,A -85,B 0,C 180,E1 -2514.656,E2 -2514.656} C_VEL
LIN {X 0,Y 565.956,Z 630.326,A -85,B 0,C 180,E1 -2515.727,E2 -2515.727} C_VEL
LIN {X 0,Y 565.876,Z 633.739,A -85,B 0,C 180,E1 -2517.152,E2 -2517.152} C_VEL
LIN {X 0,Y 565.844,Z 635.776,A -85,B 0,C 180,E1 -2518.577,E2 -2518.577} C_VEL
LIN {X 0,Y 565.836,Z 636.496,A -85,B 0,C 180,E1 -2520,E2 -2520} C_VEL
LIN {X 0,Y 565.84,Z 635.878,A -85,B 0,C 180,E1 -2521.423,E2 -2521.423} C_VEL
LIN {X 0,Y 565.875,Z 633.918,A -85,B 0,C 180,E1 -2522.847,E2 -2522.847} C_VEL
LIN {X 0,Y 565.958,Z 630.574,A -85,B 0,C 180,E1 -2524.273,E2 -2524.273} C_VEL
LIN {X 0,Y 565.985,Z 625.76,A -85,B 0,C 180,E1 -2525.701,E2 -2525.701} C_VEL
LIN {X 0,Y 565.997,Z 621.247,A -85,B 0,C 180,E1 -2526.739,E2 -2526.739} C_VEL
LIN {X 0,Y 566.045,Z 614.303,A -85,B 0,C 180,E1 -2528.029,E2 -2528.029} C_VEL
LIN {X 0,Y 566.172,Z 605.916,A -85,B 0,C 180,E1 -2529.286,E2 -2529.286} C_VEL
LIN {X 0,Y 566.283,Z 597.143,A -85,B 0,C 180,E1 -2530.367,E2 -2530.367} C_VEL
LIN {X 0,Y 566.468,Z 586.505,A -85,B 0,C 180,E1 -2531.45,E2 -2531.45} C_VEL
LIN {X 0,Y 566.617,Z 575.739,A -85,B 0,C 180,E1 -2532.354,E2 -2532.354} C_VEL
LIN {X 0,Y 566.767,Z 563.959,A -85,B 0,C 180,E1 -2533.171,E2 -2533.171} C_VEL
LIN {X 0,Y 567.027,Z 550.96,A -85,B 0,C 180,E1 -2533.895,E2 -2533.895} C_VEL
LIN {X 0,Y 567.235,Z 538.211,A -85,B 0,C 180,E1 -2534.452,E2 -2534.452} C_VEL
LIN {X 0,Y 567.313,Z 524.636,A -85,B 0,C 180,E1 -2534.901,E2 -2534.901} C_VEL
LIN {X 0,Y 567.45,Z 510.585,A -85,B 0,C 180,E1 -2535.213,E2 -2535.213} C_VEL
LIN {X 0,Y 567.664,Z 381.549,A -85,B 0,C 180,E1 -2536.885,E2 -2536.885} C_VEL
LIN {X 0,Y 566.513,Z 375.857,A -85,B 0,C 180,E1 -2537.013,E2 -2537.013} C_VEL
LIN {X 0,Y 566.48,Z 373.728,A -85,B 0,C 180,E1 -2537.323,E2 -2537.323} C_VEL
LIN {X 0,Y 566.741,Z 363.8,A -85,B 0,C 180,E1 -2539.132,E2 -2539.132} C_VEL
LIN {X 0,Y 566.223,Z 360.631,A -85,B 0,C 180,E1 -2539.769,E2 -2539.769} C_VEL
LIN {X 0,Y 566.181,Z 360.588,A -85,B 0,C 180,E1 -2542.631,E2 -2542.631} C_VEL
LIN {X 0,Y 566.223,Z 360.581,A -85,B 0,C 180,E1 -2545.03,E2 -2545.03} C_VEL
LIN {X 0,Y 566.212,Z 360.578,A -85,B 0,C 180,E1 -2547.339,E2 -2547.339} C_VEL
LIN {X 0,Y 566.205,Z 360.577,A -85,B 0,C 180,E1 -2549.769,E2 -2549.769} C_VEL
LIN {X 0,Y 566.207,Z 360.584,A -85,B 0,C 180,E1 -2552.429,E2 -2552.429} C_VEL
LIN {X 0,Y 566.184,Z 360.582,A -85,B 0,C 180,E1 -2554.989,E2 -2554.989} C_VEL
LIN {X 0,Y 566.195,Z 360.578,A -85,B 0,C 180,E1 -2557.461,E2 -2557.461} C_VEL
LIN {X 0,Y 566.21,Z 360.583,A -85,B 0,C 180,E1 -2560.199,E2 -2560.199} C_VEL
LIN {X 0,Y 566.19,Z 360.579,A -85,B 0,C 180,E1 -2563.055,E2 -2563.055} C_VEL
LIN {X 0,Y 566.16,Z 360.59,A -85,B 0,C 180,E1 -2566.053,E2 -2566.053} C_VEL
LIN {X 0,Y 566.159,Z 360.584,A -85,B 0,C 180,E1 -2568.858,E2 -2568.858} C_VEL
LIN {X 0,Y 566.203,Z 360.579,A -85,B 0,C 180,E1 -2571.443,E2 -2571.443} C_VEL
LIN {X 0,Y 566.138,Z 360.591,A -85,B 0,C 180,E1 -2574.305,E2 -2574.305} C_VEL
LIN {X 0,Y 566.162,Z 360.584,A -85,B 0,C 180,E1 -2576.893,E2 -2576.893} C_VEL
LIN {X 0,Y 566.201,Z 360.585,A -85,B 0,C 180,E1 -2579.82,E2 -2579.82} C_VEL
LIN {X 0,Y 566.239,Z 360.937,A -85,B 0,C 180,E1 -2580.117,E2 -2580.117} C_VEL
LIN {X 0,Y 568.918,Z 370.413,A -85,B 0,C 180,E1 -2581.097,E2 -2581.097} C_VEL
LIN {X 0,Y 568.701,Z 398.867,A -85,B 0,C 180,E1 -2583.583,E2 -2583.583} C_VEL
LIN {X 0,Y 568.203,Z 430.349,A -85,B 0,C 180,E1 -2586.395,E2 -2586.395} C_VEL
LIN {X 0,Y 567.698,Z 462.591,A -85,B 0,C 180,E1 -2589.244,E2 -2589.244} C_VEL
LIN {X 0,Y 567.622,Z 473.035,A -85,B 0,C 180,E1 -2590.128,E2 -2590.128} C_VEL
LIN {X 0,Y 568.507,Z 479.598,A -85,B 0,C 180,E1 -2590.254,E2 -2590.254} C_VEL
LIN {X 0,Y 567.987,Z 640.885,A -85,B 0,C 180,E1 -2592.363,E2 -2592.363} C_VEL
LIN {X 0,Y 567.855,Z 656.684,A -85,B 0,C 180,E1 -2592.72,E2 -2592.72} C_VEL
LIN {X 0,Y 567.606,Z 672.023,A -85,B 0,C 180,E1 -2593.222,E2 -2593.222} C_VEL
LIN {X 0,Y 567.445,Z 685.747,A -85,B 0,C 180,E1 -2593.818,E2 -2593.818} C_VEL
LIN {X 0,Y 567.153,Z 699.228,A -85,B 0,C 180,E1 -2594.548,E2 -2594.548} C_VEL
LIN {X 0,Y 566.925,Z 712.494,A -85,B 0,C 180,E1 -2595.428,E2 -2595.428} C_VEL
LIN {X 0,Y 566.675,Z 725.342,A -85,B 0,C 180,E1 -2596.461,E2 -2596.461} C_VEL
LIN {X 0,Y 566.492,Z 735.739,A -85,B 0,C 180,E1 -2597.46,E2 -2597.46} C_VEL
LIN {X 0,Y 566.27,Z 746.306,A -85,B 0,C 180,E1 -2598.658,E2 -2598.658} C_VEL
LIN {X 0,Y 566.209,Z 754.85,A -85,B 0,C 180,E1 -2599.811,E2 -2599.811} C_VEL
LIN {X 0,Y 566.058,Z 762.725,A -85,B 0,C 180,E1 -2601.071,E2 -2601.071} C_VEL
LIN {X 0,Y 565.998,Z 770.083,A -85,B 0,C 180,E1 -2602.508,E2 -2602.508} C_VEL
LIN {X 0,Y 565.957,Z 775.921,A -85,B 0,C 180,E1 -2603.94,E2 -2603.94} C_VEL
LIN {X 0,Y 565.867,Z 779.382,A -85,B 0,C 180,E1 -2605.011,E2 -2605.011} C_VEL
LIN {X 0,Y 565.91,Z 782.885,A -85,B 0,C 180,E1 -2606.439,E2 -2606.439} C_VEL
LIN {X 0,Y 565.837,Z 785.189,A -85,B 0,C 180,E1 -2607.863,E2 -2607.863} C_VEL
LIN {X 0,Y 565.838,Z 786.348,A -85,B 0,C 180,E1 -2609.287,E2 -2609.287} C_VEL
LIN {X 0,Y 565.838,Z 786.349,A -85,B 0,C 180,E1 -2610.711,E2 -2610.711} C_VEL
LIN {X 0,Y 565.836,Z 785.193,A -85,B 0,C 180,E1 -2612.134,E2 -2612.134} C_VEL
LIN {X 0,Y 565.909,Z 782.891,A -85,B 0,C 180,E1 -2613.559,E2 -2613.559} C_VEL
LIN {X 0,Y 565.866,Z 779.388,A -85,B 0,C 180,E1 -2614.986,E2 -2614.986} C_VEL
LIN {X 0,Y 565.941,Z 774.611,A -85,B 0,C 180,E1 -2616.416,E2 -2616.416} C_VEL
LIN {X 0,Y 566.015,Z 768.43,A -85,B 0,C 180,E1 -2617.849,E2 -2617.849} C_VEL
LIN {X 0,Y 566.084,Z 760.658,A -85,B 0,C 180,E1 -2619.287,E2 -2619.287} C_VEL
LIN {X 0,Y 566.238,Z 752.378,A -85,B 0,C 180,E1 -2620.548,E2 -2620.548} C_VEL
LIN {X 0,Y 566.365,Z 742.402,A -85,B 0,C 180,E1 -2621.813,E2 -2621.813} C_VEL
LIN {X 0,Y 566.584,Z 732.201,A -85,B 0,C 180,E1 -2622.9,E2 -2622.9} C_VEL
LIN {X 0,Y 566.798,Z 720.03,A -85,B 0,C 180,E1 -2623.991,E2 -2623.991} C_VEL
LIN {X 0,Y 567.037,Z 707.357,A -85,B 0,C 180,E1 -2624.935,E2 -2624.935} C_VEL
LIN {X 0,Y 567.228,Z 694.542,A -85,B 0,C 180,E1 -2625.724,E2 -2625.724} C_VEL
LIN {X 0,Y 567.514,Z 679.86,A -85,B 0,C 180,E1 -2626.455,E2 -2626.455} C_VEL
LIN {X 0,Y 567.709,Z 665.644,A -85,B 0,C 180,E1 -2627.004,E2 -2627.004} C_VEL
LIN {X 0,Y 567.9,Z 650.334,A -85,B 0,C 180,E1 -2627.441,E2 -2627.441} C_VEL
LIN {X 0,Y 568.013,Z 635.711,A -85,B 0,C 180,E1 -2627.716,E2 -2627.716} C_VEL
LIN {X 0,Y 568.49,Z 478.803,A -85,B 0,C 180,E1 -2629.757,E2 -2629.757} C_VEL
LIN {X 0,Y 567.583,Z 472.575,A -85,B 0,C 180,E1 -2629.895,E2 -2629.895} C_VEL
LIN {X 0,Y 568.076,Z 437.882,A -85,B 0,C 180,E1 -2632.935,E2 -2632.935} C_VEL
LIN {X 0,Y 568.643,Z 405.609,A -85,B 0,C 180,E1 -2635.826,E2 -2635.826} C_VEL
LIN {X 0,Y 569.023,Z 374.467,A -85,B 0,C 180,E1 -2638.591,E2 -2638.591} C_VEL
LIN {X 0,Y 568.871,Z 369.991,A -85,B 0,C 180,E1 -2639.005,E2 -2639.005} C_VEL
LIN {X 0,Y 566.203,Z 360.783,A -85,B 0,C 180,E1 -2640.023,E2 -2640.023} C_VEL
LIN {X 0,Y 566.147,Z 360.584,A -85,B 0,C 180,E1 -2641.423,E2 -2641.423} C_VEL
LIN {X 0,Y 566.183,Z 360.586,A -85,B 0,C 180,E1 -2643.956,E2 -2643.956} C_VEL
LIN {X 0,Y 566.133,Z 360.591,A -85,B 0,C 180,E1 -2646.573,E2 -2646.573} C_VEL
LIN {X 0,Y 566.193,Z 360.578,A -85,B 0,C 180,E1 -2649.273,E2 -2649.273} C_VEL
LIN {X 0,Y 566.168,Z 360.587,A -85,B 0,C 180,E1 -2652.089,E2 -2652.089} C_VEL
LIN {X 0,Y 566.145,Z 360.584,A -85,B 0,C 180,E1 -2655.036,E2 -2655.036} C_VEL
LIN {X 0,Y 566.128,Z 360.585,A -85,B 0,C 180,E1 -2658.144,E2 -2658.144} C_VEL
LIN {X 0,Y 566.191,Z 360.582,A -85,B 0,C 180,E1 -2660.724,E2 -2660.724} C_VEL
LIN {X 0,Y 566.13,Z 360.581,A -85,B 0,C 180,E1 -2663.425,E2 -2663.425} C_VEL
LIN {X 0,Y 566.181,Z 360.58,A -85,B 0,C 180,E1 -2666.268,E2 -2666.268} C_VEL
LIN {X 0,Y 566.167,Z 360.582,A -85,B 0,C 180,E1 -2668.924,E2 -2668.924} C_VEL
LIN {X 0,Y 566.132,Z 360.585,A -85,B 0,C 180,E1 -2671.853,E2 -2671.853} C_VEL
LIN {X 0,Y 566.177,Z 360.586,A -85,B 0,C 180,E1 -2674.249,E2 -2674.249} C_VEL
LIN {X 0,Y 566.144,Z 360.583,A -85,B 0,C 180,E1 -2677.367,E2 -2677.367} C_VEL
LIN {X 0,Y 566.153,Z 360.58,A -85,B 0,C 180,E1 -2679.661,E2 -2679.661} C_VEL
LIN {X 0,Y 566.148,Z 360.584,A -85,B 0,C 180,E1 -2681.92,E2 -2681.92} C_VEL
LIN {X 0,Y 566.163,Z 360.582,A -85,B 0,C 180,E1 -2684.89,E2 -2684.89} C_VEL
LIN {X 0,Y 566.156,Z 360.582,A -85,B 0,C 180,E1 -2687.817,E2 -2687.817} C_VEL
LIN {X 0,Y 566.134,Z 360.585,A -85,B 0,C 180,E1 -2689.991,E2 -2689.991} C_VEL
LIN {X 0,Y 566.168,Z 360.584,A -85,B 0,C 180,E1 -2692.869,E2 -2692.869} C_VEL
LIN {X 0,Y 566.239,Z 360.571,A -85,B 0,C 180,E1 -2695.016,E2 -2695.016} C_VEL
LIN {X 0,Y 566.242,Z 360.571,A -85,B 0,C 180,E1 -2697.866,E2 -2697.866} C_VEL
LIN {X 0,Y 566.285,Z 360.57,A -85,B 0,C 180,E1 -2700.711,E2 -2700.711} C_VEL
LIN {X 0,Y 566.245,Z 360.576,A -85,B 0,C 180,E1 -2702.846,E2 -2702.846} C_VEL
LIN {X 0,Y 566.213,Z 360.573,A -85,B 0,C 180,E1 -2705.699,E2 -2705.699} C_VEL
LIN {X 0,Y 566.167,Z 360.579,A -85,B 0,C 180,E1 -2707.848,E2 -2707.848} C_VEL
LIN {X 0,Y 566.202,Z 360.581,A -85,B 0,C 180,E1 -2710.73,E2 -2710.73} C_VEL
LIN {X 0,Y 566.159,Z 360.58,A -85,B 0,C 180,E1 -2713.642,E2 -2713.642} C_VEL
LIN {X 0,Y 566.19,Z 360.584,A -85,B 0,C 180,E1 -2716.588,E2 -2716.588} C_VEL
LIN {X 0,Y 566.183,Z 360.578,A -85,B 0,C 180,E1 -2719.582,E2 -2719.582} C_VEL
LIN {X 0,Y 566.169,Z 360.578,A -85,B 0,C 180,E1 -2721.864,E2 -2721.864} C_VEL
LIN {X 0,Y 566.132,Z 360.586,A -85,B 0,C 180,E1 -2724.397,E2 -2724.397} C_VEL
LIN {X 0,Y 566.149,Z 360.59,A -85,B 0,C 180,E1 -2726.651,E2 -2726.651} C_VEL
LIN {X 0,Y 566.138,Z 360.584,A -85,B 0,C 180,E1 -2727.495,E2 -2727.495} C_VEL
LIN {X 0,Y 565.46,Z 360.671,A -85,B 0,C 180,E1 -2728.089,E2 -2728.089} C_VEL
LIN {X 0,Y 562.587,Z 361.03,A -85,B 0,C 180,E1 -2729.053,E2 -2729.053} C_VEL
LIN {X 0,Y 560.179,Z 361.328,A -85,B 0,C 180,E1 -2729.828,E2 -2729.828} C_VEL
LIN {X 0,Y 559.165,Z 361.457,A -85,B 0,C 180,E1 -2730.427,E2 -2730.427} C_VEL
LIN {X 0,Y 559.094,Z 361.463,A -85,B 0,C 180,E1 -2730.63,E2 -2730.63} C_VEL
LIN {X 0,Y 559.133,Z 361.465,A -85,B 0,C 180,E1 -2732.717,E2 -2732.717} C_VEL
LIN {X 0,Y 559.104,Z 361.461,A -85,B 0,C 180,E1 -2735.326,E2 -2735.326} C_VEL
LIN {X 0,Y 559.107,Z 361.455,A -85,B 0,C 180,E1 -2738.02,E2 -2738.02} C_VEL
LIN {X 0,Y 559.111,Z 361.467,A -85,B 0,C 180,E1 -2740.817,E2 -2740.817} C_VEL
LIN {X 0,Y 559.092,Z 361.461,A -85,B 0,C 180,E1 -2743.739,E2 -2743.739} C_VEL
LIN {X 0,Y 559.083,Z 361.464,A -85,B 0,C 180,E1 -2746.263,E2 -2746.263} C_VEL
LIN {X 0,Y 559.104,Z 361.463,A -85,B 0,C 180,E1 -2749.185,E2 -2749.185} C_VEL
LIN {X 0,Y 559.156,Z 361.46,A -85,B 0,C 180,E1 -2751.194,E2 -2751.194} C_VEL
LIN {X 0,Y 559.1,Z 361.463,A -85,B 0,C 180,E1 -2753.788,E2 -2753.788} C_VEL
LIN {X 0,Y 559.127,Z 361.449,A -85,B 0,C 180,E1 -2756.425,E2 -2756.425} C_VEL
LIN {X 0,Y 559.134,Z 361.53,A -85,B 0,C 180,E1 -2758.845,E2 -2758.845} C_VEL
LIN {X 0,Y 559.315,Z 362.366,A -85,B 0,C 180,E1 -2758.992,E2 -2758.992} C_VEL
LIN {X 0,Y 562.183,Z 373.177,A -85,B 0,C 180,E1 -2760.205,E2 -2760.205} C_VEL
LIN {X 0,Y 561.876,Z 398.061,A -85,B 0,C 180,E1 -2762.632,E2 -2762.632} C_VEL
LIN {X 0,Y 561.5,Z 423.657,A -85,B 0,C 180,E1 -2765.112,E2 -2765.112} C_VEL
LIN {X 0,Y 560.978,Z 453.124,A -85,B 0,C 180,E1 -2767.984,E2 -2767.984} C_VEL
LIN {X 0,Y 560.662,Z 473.468,A -85,B 0,C 180,E1 -2769.916,E2 -2769.916} C_VEL
LIN {X 0,Y 561.823,Z 481.085,A -85,B 0,C 180,E1 -2770.074,E2 -2770.074} C_VEL
LIN {X 0,Y 561.244,Z 640.331,A -85,B 0,C 180,E1 -2772.182,E2 -2772.182} C_VEL
LIN {X 0,Y 561.095,Z 655.897,A -85,B 0,C 180,E1 -2772.531,E2 -2772.531} C_VEL
LIN {X 0,Y 560.866,Z 669.614,A -85,B 0,C 180,E1 -2772.97,E2 -2772.97} C_VEL
LIN {X 0,Y 560.571,Z 684.834,A -85,B 0,C 180,E1 -2773.617,E2 -2773.617} C_VEL
LIN {X 0,Y 560.286,Z 698.504,A -85,B 0,C 180,E1 -2774.356,E2 -2774.356} C_VEL
LIN {X 0,Y 560.026,Z 711.774,A -85,B 0,C 180,E1 -2775.238,E2 -2775.238} C_VEL
LIN {X 0,Y 559.706,Z 724.84,A -85,B 0,C 180,E1 -2776.291,E2 -2776.291} C_VEL
LIN {X 0,Y 559.52,Z 735.335,A -85,B 0,C 180,E1 -2777.303,E2 -2777.303} C_VEL
LIN {X 0,Y 559.315,Z 746.23,A -85,B 0,C 180,E1 -2778.55,E2 -2778.55} C_VEL
LIN {X 0,Y 559.16,Z 755.794,A -85,B 0,C 180,E1 -2779.867,E2 -2779.867} C_VEL
LIN {X 0,Y 558.995,Z 763.509,A -85,B 0,C 180,E1 -2781.142,E2 -2781.142} C_VEL
LIN {X 0,Y 558.92,Z 769.904,A -85,B 0,C 180,E1 -2782.414,E2 -2782.414} C_VEL
LIN {X 0,Y 558.859,Z 775.782,A -85,B 0,C 180,E1 -2783.865,E2 -2783.865} C_VEL
LIN {X 0,Y 558.786,Z 779.259,A -85,B 0,C 180,E1 -2784.95,E2 -2784.95} C_VEL
LIN {X 0,Y 558.818,Z 782.797,A -85,B 0,C 180,E1 -2786.396,E2 -2786.396} C_VEL
LIN {X 0,Y 558.744,Z 785.142,A -85,B 0,C 180,E1 -2787.839,E2 -2787.839} C_VEL
LIN {X 0,Y 558.737,Z 786.338,A -85,B 0,C 180,E1 -2789.28,E2 -2789.28} C_VEL
LIN {X 0,Y 558.738,Z 786.359,A -85,B 0,C 180,E1 -2790.722,E2 -2790.722} C_VEL
LIN {X 0,Y 558.745,Z 785.24,A -85,B 0,C 180,E1 -2792.164,E2 -2792.164} C_VEL
LIN {X 0,Y 558.82,Z 782.974,A -85,B 0,C 180,E1 -2793.606,E2 -2793.606} C_VEL
LIN {X 0,Y 558.786,Z 779.512,A -85,B 0,C 180,E1 -2795.052,E2 -2795.052} C_VEL
LIN {X 0,Y 558.845,Z 774.632,A -85,B 0,C 180,E1 -2796.537,E2 -2796.537} C_VEL
LIN {X 0,Y 558.942,Z 768.633,A -85,B 0,C 180,E1 -2797.951,E2 -2797.951} C_VEL
LIN {X 0,Y 559.003,Z 760.908,A -85,B 0,C 180,E1 -2799.408,E2 -2799.408} C_VEL
LIN {X 0,Y 559.215,Z 752.672,A -85,B 0,C 180,E1 -2800.684,E2 -2800.684} C_VEL
LIN {X 0,Y 559.319,Z 742.753,A -85,B 0,C 180,E1 -2801.967,E2 -2801.967} C_VEL
LIN {X 0,Y 559.57,Z 732.631,A -85,B 0,C 180,E1 -2803.067,E2 -2803.067} C_VEL
LIN {X 0,Y 559.824,Z 720.531,A -85,B 0,C 180,E1 -2804.171,E2 -2804.171} C_VEL
LIN {X 0,Y 560.133,Z 707.667,A -85,B 0,C 180,E1 -2805.146,E2 -2805.146} C_VEL
LIN {X 0,Y 560.359,Z 695.309,A -85,B 0,C 180,E1 -2805.925,E2 -2805.925} C_VEL
LIN {X 0,Y 560.66,Z 680.818,A -85,B 0,C 180,E1 -2806.664,E2 -2806.664} C_VEL
LIN {X 0,Y 560.915,Z 665.557,A -85,B 0,C 180,E1 -2807.266,E2 -2807.266} C_VEL
LIN {X 0,Y 561.112,Z 649.909,A -85,B 0,C 180,E1 -2807.715,E2 -2807.715} C_VEL
LIN {X 0,Y 561.274,Z 634.182,A -85,B 0,C 180,E1 -2808.006,E2 -2808.006} C_VEL
LIN {X 0,Y 561.744,Z 480.262,A -85,B 0,C 180,E1 -2810.03,E2 -2810.03} C_VEL
LIN {X 0,Y 560.675,Z 473.127,A -85,B 0,C 180,E1 -2810.191,E2 -2810.191} C_VEL
LIN {X 0,Y 561.113,Z 443.498,A -85,B 0,C 180,E1 -2813.043,E2 -2813.043} C_VEL
LIN {X 0,Y 561.652,Z 415.987,A -85,B 0,C 180,E1 -2815.718,E2 -2815.718} C_VEL
LIN {X 0,Y 562.055,Z 385.83,A -85,B 0,C 180,E1 -2818.648,E2 -2818.648} C_VEL
LIN {X 0,Y 562.184,Z 372.99,A -85,B 0,C 180,E1 -2819.901,E2 -2819.901} C_VEL
LIN {X 0,Y 559.142,Z 361.669,A -85,B 0,C 180,E1 -2821.199,E2 -2821.199} C_VEL
LIN {X 0,Y 559.104,Z 361.457,A -85,B 0,C 180,E1 -2823.939,E2 -2823.939} C_VEL
LIN {X 0,Y 559.097,Z 361.467,A -85,B 0,C 180,E1 -2827.113,E2 -2827.113} C_VEL
LIN {X 0,Y 559.118,Z 361.46,A -85,B 0,C 180,E1 -2829.936,E2 -2829.936} C_VEL
LIN {X 0,Y 559.11,Z 361.46,A -85,B 0,C 180,E1 -2832.749,E2 -2832.749} C_VEL
LIN {X 0,Y 559.109,Z 361.459,A -85,B 0,C 180,E1 -2835.766,E2 -2835.766} C_VEL
LIN {X 0,Y 559.095,Z 361.462,A -85,B 0,C 180,E1 -2838.223,E2 -2838.223} C_VEL
LIN {X 0,Y 559.139,Z 361.46,A -85,B 0,C 180,E1 -2841.063,E2 -2841.063} C_VEL
LIN {X 0,Y 559.115,Z 361.458,A -85,B 0,C 180,E1 -2843.787,E2 -2843.787} C_VEL
LIN {X 0,Y 559.126,Z 361.455,A -85,B 0,C 180,E1 -2846.423,E2 -2846.423} C_VEL
LIN {X 0,Y 559.144,Z 361.463,A -85,B 0,C 180,E1 -2848.98,E2 -2848.98} C_VEL
LIN {X 0,Y 559.113,Z 361.462,A -85,B 0,C 180,E1 -2851.63,E2 -2851.63} C_VEL
LIN {X 0,Y 559.143,Z 361.457,A -85,B 0,C 180,E1 -2853.901,E2 -2853.901} C_VEL
LIN {X 0,Y 559.114,Z 361.469,A -85,B 0,C 180,E1 -2857.066,E2 -2857.066} C_VEL
LIN {X 0,Y 559.175,Z 361.46,A -85,B 0,C 180,E1 -2859.395,E2 -2859.395} C_VEL
LIN {X 0,Y 559.189,Z 361.617,A -85,B 0,C 180,E1 -2860.347,E2 -2860.347} C_VEL
LIN {X 0,Y 559.729,Z 365.876,A -85,B 0,C 180,E1 -2861.136,E2 -2861.136} C_VEL
LIN {X 0,Y 559.553,Z 374.705,A -85,B 0,C 180,E1 -2862.663,E2 -2862.663} C_VEL
LIN {X 0,Y 559.75,Z 377.187,A -85,B 0,C 180,E1 -2862.892,E2 -2862.892} C_VEL
LIN {X 0,Y 560.981,Z 383.862,A -85,B 0,C 180,E1 -2863.022,E2 -2863.022} C_VEL
LIN {X 0,Y 560.58,Z 511.983,A -85,B 0,C 180,E1 -2864.712,E2 -2864.712} C_VEL
LIN {X 0,Y 560.456,Z 526.56,A -85,B 0,C 180,E1 -2865.061,E2 -2865.061} C_VEL
LIN {X 0,Y 560.242,Z 540.941,A -85,B 0,C 180,E1 -2865.562,E2 -2865.562} C_VEL
LIN {X 0,Y 560.05,Z 554.553,A -85,B 0,C 180,E1 -2866.206,E2 -2866.206} C_VEL
LIN {X 0,Y 559.809,Z 566.809,A -85,B 0,C 180,E1 -2866.94,E2 -2866.94} C_VEL
LIN {X 0,Y 559.564,Z 579.205,A -85,B 0,C 180,E1 -2867.856,E2 -2867.856} C_VEL
LIN {X 0,Y 559.424,Z 590.331,A -85,B 0,C 180,E1 -2868.866,E2 -2868.866} C_VEL
LIN {X 0,Y 559.198,Z 599.483,A -85,B 0,C 180,E1 -2869.866,E2 -2869.866} C_VEL
LIN {X 0,Y 559.079,Z 609.107,A -85,B 0,C 180,E1 -2871.142,E2 -2871.142} C_VEL
LIN {X 0,Y 558.968,Z 616.91,A -85,B 0,C 180,E1 -2872.414,E2 -2872.414} C_VEL
LIN {X 0,Y 558.875,Z 622.343,A -85,B 0,C 180,E1 -2873.501,E2 -2873.501} C_VEL
LIN {X 0,Y 558.859,Z 626.779,A -85,B 0,C 180,E1 -2874.588,E2 -2874.588} C_VEL
LIN {X 0,Y 558.866,Z 630.325,A -85,B 0,C 180,E1 -2875.673,E2 -2875.673} C_VEL
LIN {X 0,Y 558.797,Z 633.738,A -85,B 0,C 180,E1 -2877.116,E2 -2877.116} C_VEL
LIN {X 0,Y 558.743,Z 635.775,A -85,B 0,C 180,E1 -2878.558,E2 -2878.558} C_VEL
LIN {X 0,Y 558.736,Z 636.496,A -85,B 0,C 180,E1 -2880,E2 -2880} C_VEL
LIN {X 0,Y 558.74,Z 635.878,A -85,B 0,C 180,E1 -2881.441,E2 -2881.441} C_VEL
LIN {X 0,Y 558.797,Z 633.916,A -85,B 0,C 180,E1 -2882.884,E2 -2882.884} C_VEL
LIN {X 0,Y 558.867,Z 630.571,A -85,B 0,C 180,E1 -2884.327,E2 -2884.327} C_VEL
LIN {X 0,Y 558.914,Z 625.755,A -85,B 0,C 180,E1 -2885.773,E2 -2885.773} C_VEL
LIN {X 0,Y 558.905,Z 621.069,A -85,B 0,C 180,E1 -2886.86,E2 -2886.86} C_VEL
LIN {X 0,Y 558.986,Z 614.296,A -85,B 0,C 180,E1 -2888.131,E2 -2888.131} C_VEL
LIN {X 0,Y 559.107,Z 605.908,A -85,B 0,C 180,E1 -2889.405,E2 -2889.405} C_VEL
LIN {X 0,Y 559.265,Z 597.137,A -85,B 0,C 180,E1 -2890.499,E2 -2890.499} C_VEL
LIN {X 0,Y 559.451,Z 586.494,A -85,B 0,C 180,E1 -2891.595,E2 -2891.595} C_VEL
LIN {X 0,Y 559.63,Z 575.725,A -85,B 0,C 180,E1 -2892.511,E2 -2892.511} C_VEL
LIN {X 0,Y 559.814,Z 563.944,A -85,B 0,C 180,E1 -2893.337,E2 -2893.337} C_VEL
LIN {X 0,Y 560.108,Z 550.943,A -85,B 0,C 180,E1 -2894.07,E2 -2894.07} C_VEL
LIN {X 0,Y 560.355,Z 538.46,A -85,B 0,C 180,E1 -2894.623,E2 -2894.623} C_VEL
LIN {X 0,Y 560.46,Z 524.484,A -85,B 0,C 180,E1 -2895.091,E2 -2895.091} C_VEL
LIN {X 0,Y 560.604,Z 510.545,A -85,B 0,C 180,E1 -2895.404,E2 -2895.404} C_VEL
LIN {X 0,Y 561.001,Z 383.17,A -85,B 0,C 180,E1 -2897.083,E2 -2897.083} C_VEL
LIN {X 0,Y 559.689,Z 376.645,A -85,B 0,C 180,E1 -2897.251,E2 -2897.251} C_VEL
LIN {X 0,Y 559.799,Z 371.672,A -85,B 0,C 180,E1 -2898.103,E2 -2898.103} C_VEL
LIN {X 0,Y 559.903,Z 365.455,A -85,B 0,C 180,E1 -2899.25,E2 -2899.25} C_VEL
LIN {X 0,Y 559.178,Z 361.502,A -85,B 0,C 180,E1 -2900.029,E2 -2900.029} C_VEL
LIN {X 0,Y 559.143,Z 361.461,A -85,B 0,C 180,E1 -2902.153,E2 -2902.153} C_VEL
LIN {X 0,Y 559.181,Z 361.456,A -85,B 0,C 180,E1 -2905.298,E2 -2905.298} C_VEL
LIN {X 0,Y 559.152,Z 361.456,A -85,B 0,C 180,E1 -2907.714,E2 -2907.714} C_VEL
LIN {X 0,Y 559.157,Z 361.459,A -85,B 0,C 180,E1 -2910.182,E2 -2910.182} C_VEL
LIN {X 0,Y 559.161,Z 361.462,A -85,B 0,C 180,E1 -2912.715,E2 -2912.715} C_VEL
LIN {X 0,Y 559.128,Z 361.459,A -85,B 0,C 180,E1 -2915.324,E2 -2915.324} C_VEL
LIN {X 0,Y 559.133,Z 361.462,A -85,B 0,C 180,E1 -2918.018,E2 -2918.018} C_VEL
LIN {X 0,Y 559.158,Z 361.458,A -85,B 0,C 180,E1 -2920.812,E2 -2920.812} C_VEL
LIN {X 0,Y 559.114,Z 361.463,A -85,B 0,C 180,E1 -2923.737,E2 -2923.737} C_VEL
LIN {X 0,Y 559.111,Z 361.469,A -85,B 0,C 180,E1 -2926.262,E2 -2926.262} C_VEL
LIN {X 0,Y 559.121,Z 361.46,A -85,B 0,C 180,E1 -2928.954,E2 -2928.954} C_VEL
LIN {X 0,Y 559.171,Z 361.454,A -85,B 0,C 180,E1 -2931.192,E2 -2931.192} C_VEL
LIN {X 0,Y 559.113,Z 361.467,A -85,B 0,C 180,E1 -2933.786,E2 -2933.786} C_VEL
LIN {X 0,Y 559.125,Z 361.464,A -85,B 0,C 180,E1 -2936.422,E2 -2936.422} C_VEL
LIN {X 0,Y 559.119,Z 361.468,A -85,B 0,C 180,E1 -2939.397,E2 -2939.397} C_VEL
LIN {X 0,Y 559.225,Z 361.808,A -85,B 0,C 180,E1 -2939.88,E2 -2939.88} C_VEL
LIN {X 0,Y 562.166,Z 373.162,A -85,B 0,C 180,E1 -2941.059,E2 -2941.059} C_VEL
LIN {X 0,Y 561.887,Z 404.625,A -85,B 0,C 180,E1 -2943.838,E2 -2943.838} C_VEL
LIN {X 0,Y 561.457,Z 432.41,A -85,B 0,C 180,E1 -2946.282,E2 -2946.282} C_VEL
LIN {X 0,Y 560.846,Z 464.742,A -85,B 0,C 180,E1 -2949.171,E2 -2949.171} C_VEL
LIN {X 0,Y 560.76,Z 472.73,A -85,B 0,C 180,E1 -2949.861,E2 -2949.861} C_VEL
LIN {X 0,Y 561.828,Z 480.267,A -85,B 0,C 180,E1 -2950.019,E2 -2950.019} C_VEL
LIN {X 0,Y 561.219,Z 640.66,A -85,B 0,C 180,E1 -2952.139,E2 -2952.139} C_VEL
LIN {X 0,Y 561.098,Z 656.684,A -85,B 0,C 180,E1 -2952.505,E2 -2952.505} C_VEL
LIN {X 0,Y 560.8,Z 672.022,A -85,B 0,C 180,E1 -2953.012,E2 -2953.012} C_VEL
LIN {X 0,Y 560.621,Z 685.749,A -85,B 0,C 180,E1 -2953.616,E2 -2953.616} C_VEL
LIN {X 0,Y 560.289,Z 699.23,A -85,B 0,C 180,E1 -2954.353,E2 -2954.353} C_VEL
LIN {X 0,Y 560.003,Z 712.278,A -85,B 0,C 180,E1 -2955.228,E2 -2955.228} C_VEL
LIN {X 0,Y 559.723,Z 724.284,A -85,B 0,C 180,E1 -2956.197,E2 -2956.197} C_VEL
LIN {X 0,Y 559.517,Z 735.74,A -85,B 0,C 180,E1 -2957.301,E2 -2957.301} C_VEL
LIN {X 0,Y 559.306,Z 745.382,A -85,B 0,C 180,E1 -2958.401,E2 -2958.401} C_VEL
LIN {X 0,Y 559.169,Z 754.849,A -85,B 0,C 180,E1 -2959.681,E2 -2959.681} C_VEL
LIN {X 0,Y 559.004,Z 762.725,A -85,B 0,C 180,E1 -2960.957,E2 -2960.957} C_VEL
LIN {X 0,Y 558.921,Z 770.083,A -85,B 0,C 180,E1 -2962.412,E2 -2962.412} C_VEL
LIN {X 0,Y 558.839,Z 775.307,A -85,B 0,C 180,E1 -2963.683,E2 -2963.683} C_VEL
LIN {X 0,Y 558.787,Z 779.383,A -85,B 0,C 180,E1 -2964.948,E2 -2964.948} C_VEL
LIN {X 0,Y 558.819,Z 782.884,A -85,B 0,C 180,E1 -2966.394,E2 -2966.394} C_VEL
LIN {X 0,Y 558.742,Z 785.188,A -85,B 0,C 180,E1 -2967.836,E2 -2967.836} C_VEL
LIN {X 0,Y 558.739,Z 786.348,A -85,B 0,C 180,E1 -2969.278,E2 -2969.278} C_VEL
LIN {X 0,Y 558.739,Z 786.349,A -85,B 0,C 180,E1 -2970.72,E2 -2970.72} C_VEL
LIN {X 0,Y 558.742,Z 785.193,A -85,B 0,C 180,E1 -2972.161,E2 -2972.161} C_VEL
LIN {X 0,Y 558.818,Z 782.891,A -85,B 0,C 180,E1 -2973.604,E2 -2973.604} C_VEL
LIN {X 0,Y 558.787,Z 779.389,A -85,B 0,C 180,E1 -2975.05,E2 -2975.05} C_VEL
LIN {X 0,Y 558.849,Z 774.611,A -85,B 0,C 180,E1 -2976.498,E2 -2976.498} C_VEL
LIN {X 0,Y 558.95,Z 768.43,A -85,B 0,C 180,E1 -2977.949,E2 -2977.949} C_VEL
LIN {X 0,Y 559.031,Z 760.658,A -85,B 0,C 180,E1 -2979.405,E2 -2979.405} C_VEL
LIN {X 0,Y 559.216,Z 752.378,A -85,B 0,C 180,E1 -2980.682,E2 -2980.682} C_VEL
LIN {X 0,Y 559.36,Z 742.402,A -85,B 0,C 180,E1 -2981.964,E2 -2981.964} C_VEL
LIN {X 0,Y 559.595,Z 732.2,A -85,B 0,C 180,E1 -2983.064,E2 -2983.064} C_VEL
LIN {X 0,Y 559.859,Z 720.029,A -85,B 0,C 180,E1 -2984.168,E2 -2984.168} C_VEL
LIN {X 0,Y 560.121,Z 707.706,A -85,B 0,C 180,E1 -2985.099,E2 -2985.099} C_VEL
LIN {X 0,Y 560.357,Z 694.54,A -85,B 0,C 180,E1 -2985.922,E2 -2985.922} C_VEL
LIN {X 0,Y 560.673,Z 679.858,A -85,B 0,C 180,E1 -2986.661,E2 -2986.661} C_VEL
LIN {X 0,Y 560.925,Z 664.332,A -85,B 0,C 180,E1 -2987.263,E2 -2987.263} C_VEL
LIN {X 0,Y 561.171,Z 648.357,A -85,B 0,C 180,E1 -2987.705,E2 -2987.705} C_VEL
LIN {X 0,Y 561.296,Z 633.057,A -85,B 0,C 180,E1 -2987.976,E2 -2987.976} C_VEL
LIN {X 0,Y 561.833,Z 479.769,A -85,B 0,C 180,E1 -2989.988,E2 -2989.988} C_VEL
LIN {X 0,Y 560.765,Z 472.789,A -85,B 0,C 180,E1 -2990.136,E2 -2990.136} C_VEL
LIN {X 0,Y 561.303,Z 440.033,A -85,B 0,C 180,E1 -2993.032,E2 -2993.032} C_VEL
LIN {X 0,Y 561.745,Z 413.097,A -85,B 0,C 180,E1 -2995.436,E2 -2995.436} C_VEL
LIN {X 0,Y 562.282,Z 380.49,A -85,B 0,C 180,E1 -2998.355,E2 -2998.355} C_VEL
LIN {X 0,Y 562.393,Z 373.587,A -85,B 0,C 180,E1 -2998.983,E2 -2998.983} C_VEL
LIN {X 0,Y 559.196,Z 361.674,A -85,B 0,C 180,E1 -3000.296,E2 -3000.296} C_VEL
LIN {X 0,Y 559.138,Z 361.463,A -85,B 0,C 180,E1 -3002.715,E2 -3002.715} C_VEL
LIN {X 0,Y 559.103,Z 361.462,A -85,B 0,C 180,E1 -3005.324,E2 -3005.324} C_VEL
LIN {X 0,Y 559.112,Z 361.466,A -85,B 0,C 180,E1 -3008.017,E2 -3008.017} C_VEL
LIN {X 0,Y 559.114,Z 361.462,A -85,B 0,C 180,E1 -3010.814,E2 -3010.814} C_VEL
LIN {X 0,Y 559.117,Z 361.459,A -85,B 0,C 180,E1 -3013.193,E2 -3013.193} C_VEL
LIN {X 0,Y 559.101,Z 361.463,A -85,B 0,C 180,E1 -3015.764,E2 -3015.764} C_VEL
LIN {X 0,Y 559.086,Z 361.462,A -85,B 0,C 180,E1 -3018.223,E2 -3018.223} C_VEL
LIN {X 0,Y 559.153,Z 361.455,A -85,B 0,C 180,E1 -3021.064,E2 -3021.064} C_VEL
LIN {X 0,Y 559.1,Z 361.458,A -85,B 0,C 180,E1 -3023.786,E2 -3023.786} C_VEL
LIN {X 0,Y 559.132,Z 361.46,A -85,B 0,C 180,E1 -3026.423,E2 -3026.423} C_VEL
LIN {X 0,Y 559.132,Z 361.458,A -85,B 0,C 180,E1 -3028.979,E2 -3028.979} C_VEL
LIN {X 0,Y 559.093,Z 361.46,A -85,B 0,C 180,E1 -3031.629,E2 -3031.629} C_VEL
LIN {X 0,Y 559.141,Z 361.458,A -85,B 0,C 180,E1 -3033.901,E2 -3033.901} C_VEL
LIN {X 0,Y 559.094,Z 361.463,A -85,B 0,C 180,E1 -3037.065,E2 -3037.065} C_VEL
LIN {X 0,Y 559.132,Z 361.454,A -85,B 0,C 180,E1 -3039.394,E2 -3039.394} C_VEL
LIN {X 0,Y 559.099,Z 361.46,A -85,B 0,C 180,E1 -3041.684,E2 -3041.684} C_VEL
LIN {X 0,Y 559.112,Z 361.463,A -85,B 0,C 180,E1 -3044.694,E2 -3044.694} C_VEL
LIN {X 0,Y 559.125,Z 361.458,A -85,B 0,C 180,E1 -3047.662,E2 -3047.662} C_VEL
LIN {X 0,Y 559.096,Z 361.46,A -85,B 0,C 180,E1 -3049.864,E2 -3049.864} C_VEL
LIN {X 0,Y 559.157,Z 361.455,A -85,B 0,C 180,E1 -3052.053,E2 -3052.053} C_VEL
LIN {X 0,Y 559.215,Z 361.446,A -85,B 0,C 180,E1 -3054.953,E2 -3054.953} C_VEL
LIN {X 0,Y 559.215,Z 361.446,A -85,B 0,C 180,E1 -3057.839,E2 -3057.839} C_VEL
LIN {X 0,Y 559.255,Z 361.445,A -85,B 0,C 180,E1 -3060.72,E2 -3060.72} C_VEL
LIN {X 0,Y 559.209,Z 361.452,A -85,B 0,C 180,E1 -3062.882,E2 -3062.882} C_VEL
LIN {X 0,Y 559.185,Z 361.449,A -85,B 0,C 180,E1 -3065.771,E2 -3065.771} C_VEL
LIN {X 0,Y 559.144,Z 361.464,A -85,B 0,C 180,E1 -3068.675,E2 -3068.675} C_VEL
LIN {X 0,Y 559.184,Z 361.446,A -85,B 0,C 180,E1 -3071.601,E2 -3071.601} C_VEL
LIN {X 0,Y 559.164,Z 361.461,A -85,B 0,C 180,E1 -3074.588,E2 -3074.588} C_VEL
LIN {X 0,Y 559.118,Z 361.457,A -85,B 0,C 180,E1 -3077.558,E2 -3077.558} C_VEL
LIN {X 0,Y 559.147,Z 361.454,A -85,B 0,C 180,E1 -3079.838,E2 -3079.838} C_VEL
LIN {X 0,Y 559.118,Z 361.459,A -85,B 0,C 180,E1 -3082.154,E2 -3082.154} C_VEL
LIN {X 0,Y 559.121,Z 361.459,A -85,B 0,C 180,E1 -3085.178,E2 -3085.178} C_VEL
LIN {X 0,Y 559.099,Z 361.461,A -85,B 0,C 180,E1 -3087.717,E2 -3087.717} C_VEL
LIN {X 0,Y 559.094,Z 361.463,A -85,B 0,C 180,E1 -3090.63,E2 -3090.63} C_VEL
LIN {X 0,Y 558.454,Z 361.546,A -85,B 0,C 180,E1 -3091.232,E2 -3091.232} C_VEL
LIN {X 0,Y 555.6,Z 361.9,A -85,B 0,C 180,E1 -3092.208,E2 -3092.208} C_VEL
LIN {X 0,Y 553.179,Z 362.205,A -85,B 0,C 180,E1 -3092.994,E2 -3092.994} C_VEL
LIN {X 0,Y 552.15,Z 362.328,A -85,B 0,C 180,E1 -3093.601,E2 -3093.601} C_VEL
LIN {X 0,Y 552.073,Z 362.337,A -85,B 0,C 180,E1 -3093.806,E2 -3093.806} C_VEL
LIN {X 0,Y 552.082,Z 362.337,A -85,B 0,C 180,E1 -3096.749,E2 -3096.749} C_VEL
LIN {X 0,Y 552.094,Z 362.335,A -85,B 0,C 180,E1 -3099.53,E2 -3099.53} C_VEL
LIN {X 0,Y 552.07,Z 362.338,A -85,B 0,C 180,E1 -3102.431,E2 -3102.431} C_VEL
LIN {X 0,Y 552.056,Z 362.338,A -85,B 0,C 180,E1 -3105.561,E2 -3105.561} C_VEL
LIN {X 0,Y 552.047,Z 362.346,A -85,B 0,C 180,E1 -3108.55,E2 -3108.55} C_VEL
LIN {X 0,Y 552.099,Z 362.337,A -85,B 0,C 180,E1 -3111.412,E2 -3111.412} C_VEL
LIN {X 0,Y 552.05,Z 362.347,A -85,B 0,C 180,E1 -3114.564,E2 -3114.564} C_VEL
LIN {X 0,Y 552.089,Z 362.326,A -85,B 0,C 180,E1 -3117.158,E2 -3117.158} C_VEL
LIN {X 0,Y 552.105,Z 362.535,A -85,B 0,C 180,E1 -3118.599,E2 -3118.599} C_VEL
LIN {X 0,Y 555.464,Z 374.809,A -85,B 0,C 180,E1 -3120.03,E2 -3120.03} C_VEL
LIN {X 0,Y 555.117,Z 400.319,A -85,B 0,C 180,E1 -3122.545,E2 -3122.545} C_VEL
LIN {X 0,Y 554.711,Z 425.288,A -85,B 0,C 180,E1 -3124.987,E2 -3124.987} C_VEL
LIN {X 0,Y 554.152,Z 455.562,A -85,B 0,C 180,E1 -3127.94,E2 -3127.94} C_VEL
LIN {X 0,Y 553.84,Z 473.234,A -85,B 0,C 180,E1 -3129.645,E2 -3129.645} C_VEL
LIN {X 0,Y 555.155,Z 481.827,A -85,B 0,C 180,E1 -3129.834,E2 -3129.834} C_VEL
LIN {X 0,Y 554.489,Z 640.313,A -85,B 0,C 180,E1 -3131.957,E2 -3131.957} C_VEL
LIN {X 0,Y 554.295,Z 655.057,A -85,B 0,C 180,E1 -3132.285,E2 -3132.285} C_VEL
LIN {X 0,Y 554.069,Z 669.621,A -85,B 0,C 180,E1 -3132.754,E2 -3132.754} C_VEL
LIN {X 0,Y 553.794,Z 682.933,A -85,B 0,C 180,E1 -3133.315,E2 -3133.315} C_VEL
LIN {X 0,Y 553.446,Z 696.978,A -85,B 0,C 180,E1 -3134.063,E2 -3134.063} C_VEL
LIN {X 0,Y 553.147,Z 710.203,A -85,B 0,C 180,E1 -3134.932,E2 -3134.932} C_VEL
LIN {X 0,Y 552.863,Z 722.755,A -85,B 0,C 180,E1 -3135.931,E2 -3135.931} C_VEL
LIN {X 0,Y 552.606,Z 733.578,A -85,B 0,C 180,E1 -3136.955,E2 -3136.955} C_VEL
LIN {X 0,Y 552.332,Z 743.575,A -85,B 0,C 180,E1 -3138.068,E2 -3138.068} C_VEL
LIN {X 0,Y 552.155,Z 753.346,A -85,B 0,C 180,E1 -3139.366,E2 -3139.366} C_VEL
LIN {X 0,Y 551.964,Z 761.475,A -85,B 0,C 180,E1 -3140.658,E2 -3140.658} C_VEL
LIN {X 0,Y 551.877,Z 768.202,A -85,B 0,C 180,E1 -3141.949,E2 -3141.949} C_VEL
LIN {X 0,Y 551.768,Z 774.619,A -85,B 0,C 180,E1 -3143.466,E2 -3143.466} C_VEL
LIN {X 0,Y 551.712,Z 779.26,A -85,B 0,C 180,E1 -3144.885,E2 -3144.885} C_VEL
LIN {X 0,Y 551.73,Z 782.799,A -85,B 0,C 180,E1 -3146.35,E2 -3146.35} C_VEL
LIN {X 0,Y 551.654,Z 785.142,A -85,B 0,C 180,E1 -3147.811,E2 -3147.811} C_VEL
LIN {X 0,Y 551.637,Z 786.338,A -85,B 0,C 180,E1 -3149.271,E2 -3149.271} C_VEL
LIN {X 0,Y 551.638,Z 786.359,A -85,B 0,C 180,E1 -3150.731,E2 -3150.731} C_VEL
LIN {X 0,Y 551.655,Z 785.239,A -85,B 0,C 180,E1 -3152.191,E2 -3152.191} C_VEL
LIN {X 0,Y 551.732,Z 782.973,A -85,B 0,C 180,E1 -3153.653,E2 -3153.653} C_VEL
LIN {X 0,Y 551.712,Z 779.51,A -85,B 0,C 180,E1 -3155.117,E2 -3155.117} C_VEL
LIN {X 0,Y 551.782,Z 774.77,A -85,B 0,C 180,E1 -3156.583,E2 -3156.583} C_VEL
LIN {X 0,Y 551.87,Z 768.628,A -85,B 0,C 180,E1 -3158.054,E2 -3158.054} C_VEL
LIN {X 0,Y 551.948,Z 760.902,A -85,B 0,C 180,E1 -3159.529,E2 -3159.529} C_VEL
LIN {X 0,Y 552.169,Z 752.665,A -85,B 0,C 180,E1 -3160.822,E2 -3160.822} C_VEL
LIN {X 0,Y 552.326,Z 742.745,A -85,B 0,C 180,E1 -3162.121,E2 -3162.121} C_VEL
LIN {X 0,Y 552.606,Z 732.625,A -85,B 0,C 180,E1 -3163.235,E2 -3163.235} C_VEL
LIN {X 0,Y 552.88,Z 720.52,A -85,B 0,C 180,E1 -3164.353,E2 -3164.353} C_VEL
LIN {X 0,Y 553.24,Z 707.85,A -85,B 0,C 180,E1 -3165.326,E2 -3165.326} C_VEL
LIN {X 0,Y 553.508,Z 695.303,A -85,B 0,C 180,E1 -3166.127,E2 -3166.127} C_VEL
LIN {X 0,Y 553.849,Z 680.804,A -85,B 0,C 180,E1 -3166.875,E2 -3166.875} C_VEL
LIN {X 0,Y 554.133,Z 665.528,A -85,B 0,C 180,E1 -3167.484,E2 -3167.484} C_VEL
LIN {X 0,Y 554.345,Z 649.951,A -85,B 0,C 180,E1 -3167.936,E2 -3167.936} C_VEL
LIN {X 0,Y 554.529,Z 634.551,A -85,B 0,C 180,E1 -3168.227,E2 -3168.227} C_VEL
LIN {X 0,Y 555.106,Z 481.137,A -85,B 0,C 180,E1 -3170.267,E2 -3170.267} C_VEL
LIN {X 0,Y 553.834,Z 473.18,A -85,B 0,C 180,E1 -3170.448,E2 -3170.448} C_VEL
LIN {X 0,Y 554.41,Z 441.378,A -85,B 0,C 180,E1 -3173.536,E2 -3173.536} C_VEL
LIN {X 0,Y 554.912,Z 414.213,A -85,B 0,C 180,E1 -3176.184,E2 -3176.184} C_VEL
LIN {X 0,Y 555.378,Z 385.195,A -85,B 0,C 180,E1 -3179.034,E2 -3179.034} C_VEL
LIN {X 0,Y 555.364,Z 374.419,A -85,B 0,C 180,E1 -3180.105,E2 -3180.105} C_VEL
LIN {X 0,Y 552.092,Z 362.513,A -85,B 0,C 180,E1 -3181.497,E2 -3181.497} C_VEL
LIN {X 0,Y 552.052,Z 362.335,A -85,B 0,C 180,E1 -3184.158,E2 -3184.158} C_VEL
LIN {X 0,Y 552.048,Z 362.343,A -85,B 0,C 180,E1 -3186.752,E2 -3186.752} C_VEL
LIN {X 0,Y 552.07,Z 362.342,A -85,B 0,C 180,E1 -3189.533,E2 -3189.533} C_VEL
LIN {X 0,Y 552.082,Z 362.332,A -85,B 0,C 180,E1 -3192.431,E2 -3192.431} C_VEL
LIN {X 0,Y 552.062,Z 362.339,A -85,B 0,C 180,E1 -3195.559,E2 -3195.559} C_VEL
LIN {X 0,Y 552.054,Z 362.34,A -85,B 0,C 180,E1 -3198.548,E2 -3198.548} C_VEL
LIN {X 0,Y 552.086,Z 362.341,A -85,B 0,C 180,E1 -3201.408,E2 -3201.408} C_VEL
LIN {X 0,Y 552.064,Z 362.336,A -85,B 0,C 180,E1 -3204.563,E2 -3204.563} C_VEL
LIN {X 0,Y 552.099,Z 362.34,A -85,B 0,C 180,E1 -3207.157,E2 -3207.157} C_VEL
LIN {X 0,Y 552.078,Z 362.336,A -85,B 0,C 180,E1 -3209.957,E2 -3209.957} C_VEL
LIN {X 0,Y 552.079,Z 362.343,A -85,B 0,C 180,E1 -3213.013,E2 -3213.013} C_VEL
LIN {X 0,Y 552.073,Z 362.338,A -85,B 0,C 180,E1 -3215.96,E2 -3215.96} C_VEL
LIN {X 0,Y 552.119,Z 362.339,A -85,B 0,C 180,E1 -3219.12,E2 -3219.12} C_VEL
LIN {X 0,Y 552.153,Z 362.467,A -85,B 0,C 180,E1 -3220.178,E2 -3220.178} C_VEL
LIN {X 0,Y 552.789,Z 367.363,A -85,B 0,C 180,E1 -3221.083,E2 -3221.083} C_VEL
LIN {X 0,Y 552.661,Z 376.361,A -85,B 0,C 180,E1 -3222.611,E2 -3222.611} C_VEL
LIN {X 0,Y 553.641,Z 381.121,A -85,B 0,C 180,E1 -3222.743,E2 -3222.743} C_VEL
LIN {X 0,Y 554.22,Z 384.242,A -85,B 0,C 180,E1 -3222.804,E2 -3222.804} C_VEL
LIN {X 0,Y 553.75,Z 511.809,A -85,B 0,C 180,E1 -3224.519,E2 -3224.519} C_VEL
LIN {X 0,Y 553.587,Z 526.159,A -85,B 0,C 180,E1 -3224.854,E2 -3224.854} C_VEL
LIN {X 0,Y 553.397,Z 540.042,A -85,B 0,C 180,E1 -3225.333,E2 -3225.333} C_VEL
LIN {X 0,Y 553.192,Z 553.147,A -85,B 0,C 180,E1 -3225.938,E2 -3225.938} C_VEL
LIN {X 0,Y 552.924,Z 565.712,A -85,B 0,C 180,E1 -3226.68,E2 -3226.68} C_VEL
LIN {X 0,Y 552.67,Z 577.099,A -85,B 0,C 180,E1 -3227.515,E2 -3227.515} C_VEL
LIN {X 0,Y 552.43,Z 587.171,A -85,B 0,C 180,E1 -3228.407,E2 -3228.407} C_VEL
LIN {X 0,Y 552.259,Z 597.941,A -85,B 0,C 180,E1 -3229.552,E2 -3229.552} C_VEL
LIN {X 0,Y 552.076,Z 606.594,A -85,B 0,C 180,E1 -3230.659,E2 -3230.659} C_VEL
LIN {X 0,Y 551.903,Z 614.844,A -85,B 0,C 180,E1 -3231.948,E2 -3231.948} C_VEL
LIN {X 0,Y 551.824,Z 620.654,A -85,B 0,C 180,E1 -3233.051,E2 -3233.051} C_VEL
LIN {X 0,Y 551.792,Z 626.778,A -85,B 0,C 180,E1 -3234.518,E2 -3234.518} C_VEL
LIN {X 0,Y 551.76,Z 630.324,A -85,B 0,C 180,E1 -3235.617,E2 -3235.617} C_VEL
LIN {X 0,Y 551.721,Z 633.736,A -85,B 0,C 180,E1 -3237.079,E2 -3237.079} C_VEL
LIN {X 0,Y 551.643,Z 635.775,A -85,B 0,C 180,E1 -3238.54,E2 -3238.54} C_VEL
LIN {X 0,Y 551.637,Z 636.496,A -85,B 0,C 180,E1 -3240,E2 -3240} C_VEL
LIN {X 0,Y 551.64,Z 635.877,A -85,B 0,C 180,E1 -3241.46,E2 -3241.46} C_VEL
LIN {X 0,Y 551.721,Z 633.914,A -85,B 0,C 180,E1 -3242.921,E2 -3242.921} C_VEL
LIN {X 0,Y 551.76,Z 630.568,A -85,B 0,C 180,E1 -3244.383,E2 -3244.383} C_VEL
LIN {X 0,Y 551.824,Z 625.751,A -85,B 0,C 180,E1 -3245.848,E2 -3245.848} C_VEL
LIN {X 0,Y 551.826,Z 621.061,A -85,B 0,C 180,E1 -3246.949,E2 -3246.949} C_VEL
LIN {X 0,Y 551.914,Z 614.289,A -85,B 0,C 180,E1 -3248.236,E2 -3248.236} C_VEL
LIN {X 0,Y 552.05,Z 605.9,A -85,B 0,C 180,E1 -3249.526,E2 -3249.526} C_VEL
LIN {X 0,Y 552.245,Z 597.128,A -85,B 0,C 180,E1 -3250.634,E2 -3250.634} C_VEL
LIN {X 0,Y 552.46,Z 586.611,A -85,B 0,C 180,E1 -3251.744,E2 -3251.744} C_VEL
LIN {X 0,Y 552.696,Z 576.008,A -85,B 0,C 180,E1 -3252.671,E2 -3252.671} C_VEL
LIN {X 0,Y 552.909,Z 564.358,A -85,B 0,C 180,E1 -3253.507,E2 -3253.507} C_VEL
LIN {X 0,Y 553.246,Z 551.421,A -85,B 0,C 180,E1 -3254.248,E2 -3254.248} C_VEL
LIN {X 0,Y 553.506,Z 539.148,A -85,B 0,C 180,E1 -3254.799,E2 -3254.799} C_VEL
LIN {X 0,Y 553.612,Z 525.717,A -85,B 0,C 180,E1 -3255.256,E2 -3255.256} C_VEL
LIN {X 0,Y 553.764,Z 511.755,A -85,B 0,C 180,E1 -3255.575,E2 -3255.575} C_VEL
LIN {X 0,Y 554.211,Z 383.429,A -85,B 0,C 180,E1 -3257.325,E2 -3257.325} C_VEL
LIN {X 0,Y 552.909,Z 377.527,A -85,B 0,C 180,E1 -3257.49,E2 -3257.49} C_VEL
LIN {X 0,Y 553.097,Z 367.505,A -85,B 0,C 180,E1 -3259.291,E2 -3259.291} C_VEL
LIN {X 0,Y 552.135,Z 362.394,A -85,B 0,C 180,E1 -3260.295,E2 -3260.295} C_VEL
LIN {X 0,Y 552.099,Z 362.34,A -85,B 0,C 180,E1 -3263.242,E2 -3263.242} C_VEL
LIN {X 0,Y 552.135,Z 362.332,A -85,B 0,C 180,E1 -3265.644,E2 -3265.644} C_VEL
LIN {X 0,Y 552.129,Z 362.338,A -85,B 0,C 180,E1 -3268.562,E2 -3268.562} C_VEL
LIN {X 0,Y 552.115,Z 362.333,A -85,B 0,C 180,E1 -3271.475,E2 -3271.475} C_VEL
LIN {X 0,Y 552.137,Z 362.334,A -85,B 0,C 180,E1 -3274.17,E2 -3274.17} C_VEL
LIN {X 0,Y 552.102,Z 362.339,A -85,B 0,C 180,E1 -3276.747,E2 -3276.747} C_VEL
LIN {X 0,Y 552.132,Z 362.331,A -85,B 0,C 180,E1 -3279.527,E2 -3279.527} C_VEL
LIN {X 0,Y 552.113,Z 362.34,A -85,B 0,C 180,E1 -3282.427,E2 -3282.427} C_VEL
LIN {X 0,Y 552.078,Z 362.338,A -85,B 0,C 180,E1 -3285.56,E2 -3285.56} C_VEL
LIN {X 0,Y 552.112,Z 362.335,A -85,B 0,C 180,E1 -3287.587,E2 -3287.587} C_VEL
LIN {X 0,Y 552.128,Z 362.335,A -85,B 0,C 180,E1 -3290.472,E2 -3290.472} C_VEL
LIN {X 0,Y 552.053,Z 362.342,A -85,B 0,C 180,E1 -3293.324,E2 -3293.324} C_VEL
LIN {X 0,Y 552.089,Z 362.344,A -85,B 0,C 180,E1 -3295.936,E2 -3295.936} C_VEL
LIN {X 0,Y 552.082,Z 362.343,A -85,B 0,C 180,E1 -3298.537,E2 -3298.537} C_VEL
LIN {X 0,Y 552.127,Z 362.546,A -85,B 0,C 180,E1 -3299.598,E2 -3299.598} C_VEL
LIN {X 0,Y 555.393,Z 375.152,A -85,B 0,C 180,E1 -3300.948,E2 -3300.948} C_VEL
LIN {X 0,Y 555.034,Z 405.797,A -85,B 0,C 180,E1 -3303.692,E2 -3303.692} C_VEL
LIN {X 0,Y 554.517,Z 439.702,A -85,B 0,C 180,E1 -3306.667,E2 -3306.667} C_VEL
LIN {X 0,Y 553.988,Z 466.893,A -85,B 0,C 180,E1 -3309.095,E2 -3309.095} C_VEL
LIN {X 0,Y 553.965,Z 472.957,A -85,B 0,C 180,E1 -3309.613,E2 -3309.613} C_VEL
LIN {X 0,Y 555.172,Z 481.232,A -85,B 0,C 180,E1 -3309.782,E2 -3309.782} C_VEL
LIN {X 0,Y 554.471,Z 641.09,A -85,B 0,C 180,E1 -3311.922,E2 -3311.922} C_VEL
LIN {X 0,Y 554.318,Z 656.685,A -85,B 0,C 180,E1 -3312.284,E2 -3312.284} C_VEL
LIN {X 0,Y 554.002,Z 672.021,A -85,B 0,C 180,E1 -3312.797,E2 -3312.797} C_VEL
LIN {X 0,Y 553.772,Z 685.751,A -85,B 0,C 180,E1 -3313.407,E2 -3313.407} C_VEL
LIN {X 0,Y 553.407,Z 699.232,A -85,B 0,C 180,E1 -3314.154,E2 -3314.154} C_VEL
LIN {X 0,Y 553.089,Z 712.281,A -85,B 0,C 180,E1 -3315.039,E2 -3315.039} C_VEL
LIN {X 0,Y 552.782,Z 724.286,A -85,B 0,C 180,E1 -3316.02,E2 -3316.02} C_VEL
LIN {X 0,Y 552.53,Z 735.74,A -85,B 0,C 180,E1 -3317.138,E2 -3317.138} C_VEL
LIN {X 0,Y 552.254,Z 746.43,A -85,B 0,C 180,E1 -3318.382,E2 -3318.382} C_VEL
LIN {X 0,Y 552.124,Z 754.847,A -85,B 0,C 180,E1 -3319.548,E2 -3319.548} C_VEL
LIN {X 0,Y 551.959,Z 762.725,A -85,B 0,C 180,E1 -3320.841,E2 -3320.841} C_VEL
LIN {X 0,Y 551.838,Z 770.083,A -85,B 0,C 180,E1 -3322.314,E2 -3322.314} C_VEL
LIN {X 0,Y 551.746,Z 775.646,A -85,B 0,C 180,E1 -3323.702,E2 -3323.702} C_VEL
LIN {X 0,Y 551.713,Z 779.383,A -85,B 0,C 180,E1 -3324.883,E2 -3324.883} C_VEL
LIN {X 0,Y 551.73,Z 782.884,A -85,B 0,C 180,E1 -3326.347,E2 -3326.347} C_VEL
LIN {X 0,Y 551.653,Z 785.187,A -85,B 0,C 180,E1 -3327.809,E2 -3327.809} C_VEL
LIN {X 0,Y 551.639,Z 786.348,A -85,B 0,C 180,E1 -3329.269,E2 -3329.269} C_VEL
LIN {X 0,Y 551.639,Z 786.349,A -85,B 0,C 180,E1 -3330.729,E2 -3330.729} C_VEL
LIN {X 0,Y 551.653,Z 785.192,A -85,B 0,C 180,E1 -3332.189,E2 -3332.189} C_VEL
LIN {X 0,Y 551.73,Z 782.891,A -85,B 0,C 180,E1 -3333.65,E2 -3333.65} C_VEL
LIN {X 0,Y 551.712,Z 779.389,A -85,B 0,C 180,E1 -3335.115,E2 -3335.115} C_VEL
LIN {X 0,Y 551.779,Z 774.611,A -85,B 0,C 180,E1 -3336.581,E2 -3336.581} C_VEL
LIN {X 0,Y 551.876,Z 768.429,A -85,B 0,C 180,E1 -3338.051,E2 -3338.051} C_VEL
LIN {X 0,Y 551.974,Z 760.657,A -85,B 0,C 180,E1 -3339.526,E2 -3339.526} C_VEL
LIN {X 0,Y 552.183,Z 752.377,A -85,B 0,C 180,E1 -3340.819,E2 -3340.819} C_VEL
LIN {X 0,Y 552.35,Z 742.402,A -85,B 0,C 180,E1 -3342.118,E2 -3342.118} C_VEL
LIN {X 0,Y 552.607,Z 732.199,A -85,B 0,C 180,E1 -3343.232,E2 -3343.232} C_VEL
LIN {X 0,Y 552.905,Z 720.029,A -85,B 0,C 180,E1 -3344.35,E2 -3344.35} C_VEL
LIN {X 0,Y 553.245,Z 707.46,A -85,B 0,C 180,E1 -3345.308,E2 -3345.308} C_VEL
LIN {X 0,Y 553.521,Z 694.538,A -85,B 0,C 180,E1 -3346.124,E2 -3346.124} C_VEL
LIN {X 0,Y 553.863,Z 679.856,A -85,B 0,C 180,E1 -3346.872,E2 -3346.872} C_VEL
LIN {X 0,Y 554.152,Z 664.331,A -85,B 0,C 180,E1 -3347.481,E2 -3347.481} C_VEL
LIN {X 0,Y 554.404,Z 648.812,A -85,B 0,C 180,E1 -3347.919,E2 -3347.919} C_VEL
LIN {X 0,Y 554.537,Z 632.552,A -85,B 0,C 180,E1 -3348.209,E2 -3348.209} C_VEL
LIN {X 0,Y 555.161,Z 481.133,A -85,B 0,C 180,E1 -3350.22,E2 -3350.22} C_VEL
LIN {X 0,Y 553.936,Z 472.682,A -85,B 0,C 180,E1 -3350.401,E2 -3350.401} C_VEL
LIN {X 0,Y 554.54,Z 440.911,A -85,B 0,C 180,E1 -3353.231,E2 -3353.231} C_VEL
LIN {X 0,Y 555.083,Z 407.767,A -85,B 0,C 180,E1 -3356.183,E2 -3356.183} C_VEL
LIN {X 0,Y 555.689,Z 375.448,A -85,B 0,C 180,E1 -3359.138,E2 -3359.138} C_VEL
LIN {X 0,Y 552.127,Z 362.523,A -85,B 0,C 180,E1 -3360.589,E2 -3360.589} C_VEL
LIN {X 0,Y 552.094,Z 362.338,A -85,B 0,C 180,E1 -3363.185,E2 -3363.185} C_VEL
LIN {X 0,Y 552.057,Z 362.343,A -85,B 0,C 180,E1 -3365.844,E2 -3365.844} C_VEL
LIN {X 0,Y 552.104,Z 362.334,A -85,B 0,C 180,E1 -3369.059,E2 -3369.059} C_VEL
LIN {X 0,Y 552.058,Z 362.339,A -85,B 0,C 180,E1 -3371.449,E2 -3371.449} C_VEL
LIN {X 0,Y 552.081,Z 362.336,A -85,B 0,C 180,E1 -3373.48,E2 -3373.48} C_VEL
LIN {X 0,Y 552.03,Z 362.34,A -85,B 0,C 180,E1 -3376.569,E2 -3376.569} C_VEL
LIN {X 0,Y 552.078,Z 362.333,A -85,B 0,C 180,E1 -3379.516,E2 -3379.516} C_VEL
LIN {X 0,Y 552.065,Z 362.344,A -85,B 0,C 180,E1 -3382.334,E2 -3382.334} C_VEL
LIN {X 0,Y 552.059,Z 362.33,A -85,B 0,C 180,E1 -3385.049,E2 -3385.049} C_VEL
LIN {X 0,Y 552.093,Z 362.333,A -85,B 0,C 180,E1 -3387.68,E2 -3387.68} C_VEL
LIN {X 0,Y 552.068,Z 362.344,A -85,B 0,C 180,E1 -3390.233,E2 -3390.233} C_VEL
LIN {X 0,Y 552.075,Z 362.337,A -85,B 0,C 180,E1 -3393.009,E2 -3393.009} C_VEL
LIN {X 0,Y 552.062,Z 362.337,A -85,B 0,C 180,E1 -3395.96,E2 -3395.96} C_VEL
LIN {X 0,Y 552.092,Z 362.342,A -85,B 0,C 180,E1 -3398.336,E2 -3398.336} C_VEL
LIN {X 0,Y 552.121,Z 362.336,A -85,B 0,C 180,E1 -3400.673,E2 -3400.673} C_VEL
LIN {X 0,Y 552.052,Z 362.339,A -85,B 0,C 180,E1 -3403.735,E2 -3403.735} C_VEL
LIN {X 0,Y 552.094,Z 362.333,A -85,B 0,C 180,E1 -3406.003,E2 -3406.003} C_VEL
LIN {X 0,Y 552.133,Z 362.329,A -85,B 0,C 180,E1 -3408.993,E2 -3408.993} C_VEL
LIN {X 0,Y 552.115,Z 362.331,A -85,B 0,C 180,E1 -3411.951,E2 -3411.951} C_VEL
LIN {X 0,Y 552.191,Z 362.322,A -85,B 0,C 180,E1 -3414.889,E2 -3414.889} C_VEL
LIN {X 0,Y 552.188,Z 362.322,A -85,B 0,C 180,E1 -3417.812,E2 -3417.812} C_VEL
LIN {X 0,Y 552.224,Z 362.32,A -85,B 0,C 180,E1 -3420.729,E2 -3420.729} C_VEL
LIN {X 0,Y 552.174,Z 362.328,A -85,B 0,C 180,E1 -3422.918,E2 -3422.918} C_VEL
LIN {X 0,Y 552.158,Z 362.324,A -85,B 0,C 180,E1 -3425.844,E2 -3425.844} C_VEL
LIN {X 0,Y 552.116,Z 362.337,A -85,B 0,C 180,E1 -3428.786,E2 -3428.786} C_VEL
LIN {X 0,Y 552.14,Z 362.323,A -85,B 0,C 180,E1 -3431.751,E2 -3431.751} C_VEL
LIN {X 0,Y 552.112,Z 362.338,A -85,B 0,C 180,E1 -3434.749,E2 -3434.749} C_VEL
LIN {X 0,Y 552.076,Z 362.334,A -85,B 0,C 180,E1 -3437.79,E2 -3437.79} C_VEL
LIN {X 0,Y 552.108,Z 362.333,A -85,B 0,C 180,E1 -3440.102,E2 -3440.102} C_VEL
LIN {X 0,Y 552.07,Z 362.34,A -85,B 0,C 180,E1 -3442.452,E2 -3442.452} C_VEL
LIN {X 0,Y 552.062,Z 362.337,A -85,B 0,C 180,E1 -3445.334,E2 -3445.334} C_VEL
LIN {X 0,Y 552.045,Z 362.341,A -85,B 0,C 180,E1 -3448.102,E2 -3448.102} C_VEL
LIN {X 0,Y 552.06,Z 362.345,A -85,B 0,C 180,E1 -3450.625,E2 -3450.625} C_VEL
LIN {X 0,Y 552.089,Z 362.338,A -85,B 0,C 180,E1 -3453.188,E2 -3453.188} C_VEL
LIN {X 0,Y 552.073,Z 362.337,A -85,B 0,C 180,E1 -3453.806,E2 -3453.806} C_VEL
LIN {X 0,Y 551.426,Z 362.424,A -85,B 0,C 180,E1 -3454.415,E2 -3454.415} C_VEL
LIN {X 0,Y 548.581,Z 362.776,A -85,B 0,C 180,E1 -3455.403,E2 -3455.403} C_VEL
LIN {X 0,Y 546.158,Z 363.076,A -85,B 0,C 180,E1 -3456.198,E2 -3456.198} C_VEL
LIN {X 0,Y 545.108,Z 363.204,A -85,B 0,C 180,E1 -3456.812,E2 -3456.812} C_VEL
LIN {X 0,Y 545.017,Z 363.212,A -85,B 0,C 180,E1 -3457.02,E2 -3457.02} C_VEL
LIN {X 0,Y 545.041,Z 363.214,A -85,B 0,C 180,E1 -3460.145,E2 -3460.145} C_VEL
LIN {X 0,Y 545.005,Z 363.221,A -85,B 0,C 180,E1 -3463.114,E2 -3463.114} C_VEL
LIN {X 0,Y 545.012,Z 363.217,A -85,B 0,C 180,E1 -3466.231,E2 -3466.231} C_VEL
LIN {X 0,Y 545.001,Z 363.225,A -85,B 0,C 180,E1 -3468.88,E2 -3468.88} C_VEL
LIN {X 0,Y 545.033,Z 363.215,A -85,B 0,C 180,E1 -3471.763,E2 -3471.763} C_VEL
LIN {X 0,Y 545.01,Z 363.224,A -85,B 0,C 180,E1 -3474.532,E2 -3474.532} C_VEL
LIN {X 0,Y 545.045,Z 363.202,A -85,B 0,C 180,E1 -3477.212,E2 -3477.212} C_VEL
LIN {X 0,Y 545.052,Z 363.331,A -85,B 0,C 180,E1 -3478.279,E2 -3478.279} C_VEL
LIN {X 0,Y 545.617,Z 365.473,A -85,B 0,C 180,E1 -3478.575,E2 -3478.575} C_VEL
LIN {X 0,Y 548.744,Z 376.765,A -85,B 0,C 180,E1 -3479.88,E2 -3479.88} C_VEL
LIN {X 0,Y 548.442,Z 399.546,A -85,B 0,C 180,E1 -3482.153,E2 -3482.153} C_VEL
LIN {X 0,Y 547.929,Z 425.926,A -85,B 0,C 180,E1 -3484.757,E2 -3484.757} C_VEL
LIN {X 0,Y 547.34,Z 456.257,A -85,B 0,C 180,E1 -3487.735,E2 -3487.735} C_VEL
LIN {X 0,Y 547.026,Z 473.237,A -85,B 0,C 180,E1 -3489.38,E2 -3489.38} C_VEL
LIN {X 0,Y 548.513,Z 483.427,A -85,B 0,C 180,E1 -3489.6,E2 -3489.6} C_VEL
LIN {X 0,Y 547.733,Z 640.463,A -85,B 0,C 180,E1 -3491.729,E2 -3491.729} C_VEL
LIN {X 0,Y 547.537,Z 655.917,A -85,B 0,C 180,E1 -3492.083,E2 -3492.083} C_VEL
LIN {X 0,Y 547.285,Z 669.629,A -85,B 0,C 180,E1 -3492.534,E2 -3492.534} C_VEL
LIN {X 0,Y 546.958,Z 682.939,A -85,B 0,C 180,E1 -3493.101,E2 -3493.101} C_VEL
LIN {X 0,Y 546.577,Z 696.983,A -85,B 0,C 180,E1 -3493.857,E2 -3493.857} C_VEL
LIN {X 0,Y 546.285,Z 709.421,A -85,B 0,C 180,E1 -3494.679,E2 -3494.679} C_VEL
LIN {X 0,Y 545.951,Z 721.705,A -85,B 0,C 180,E1 -3495.654,E2 -3495.654} C_VEL
LIN {X 0,Y 545.613,Z 733.586,A -85,B 0,C 180,E1 -3496.785,E2 -3496.785} C_VEL
LIN {X 0,Y 545.321,Z 743.581,A -85,B 0,C 180,E1 -3497.913,E2 -3497.913} C_VEL
LIN {X 0,Y 545.135,Z 753.352,A -85,B 0,C 180,E1 -3499.227,E2 -3499.227} C_VEL
LIN {X 0,Y 544.911,Z 761.476,A -85,B 0,C 180,E1 -3500.536,E2 -3500.536} C_VEL
LIN {X 0,Y 544.819,Z 768.202,A -85,B 0,C 180,E1 -3501.844,E2 -3501.844} C_VEL
LIN {X 0,Y 544.68,Z 774.992,A -85,B 0,C 180,E1 -3503.48,E2 -3503.48} C_VEL
LIN {X 0,Y 544.641,Z 779.261,A -85,B 0,C 180,E1 -3504.819,E2 -3504.819} C_VEL
LIN {X 0,Y 544.644,Z 782.799,A -85,B 0,C 180,E1 -3506.302,E2 -3506.302} C_VEL
LIN {X 0,Y 544.569,Z 785.143,A -85,B 0,C 180,E1 -3507.782,E2 -3507.782} C_VEL
LIN {X 0,Y 544.537,Z 786.338,A -85,B 0,C 180,E1 -3509.262,E2 -3509.262} C_VEL
LIN {X 0,Y 544.538,Z 786.359,A -85,B 0,C 180,E1 -3510.741,E2 -3510.741} C_VEL
LIN {X 0,Y 544.57,Z 785.239,A -85,B 0,C 180,E1 -3512.22,E2 -3512.22} C_VEL
LIN {X 0,Y 544.646,Z 782.972,A -85,B 0,C 180,E1 -3513.7,E2 -3513.7} C_VEL
LIN {X 0,Y 544.641,Z 779.508,A -85,B 0,C 180,E1 -3515.184,E2 -3515.184} C_VEL
LIN {X 0,Y 544.699,Z 774.767,A -85,B 0,C 180,E1 -3516.669,E2 -3516.669} C_VEL
LIN {X 0,Y 544.813,Z 768.624,A -85,B 0,C 180,E1 -3518.159,E2 -3518.159} C_VEL
LIN {X 0,Y 544.903,Z 760.897,A -85,B 0,C 180,E1 -3519.653,E2 -3519.653} C_VEL
LIN {X 0,Y 545.13,Z 752.658,A -85,B 0,C 180,E1 -3520.963,E2 -3520.963} C_VEL
LIN {X 0,Y 545.33,Z 742.737,A -85,B 0,C 180,E1 -3522.278,E2 -3522.278} C_VEL
LIN {X 0,Y 545.639,Z 732.617,A -85,B 0,C 180,E1 -3523.407,E2 -3523.407} C_VEL
LIN {X 0,Y 545.921,Z 720.51,A -85,B 0,C 180,E1 -3524.54,E2 -3524.54} C_VEL
LIN {X 0,Y 546.357,Z 708.28,A -85,B 0,C 180,E1 -3525.493,E2 -3525.493} C_VEL
LIN {X 0,Y 546.672,Z 695.296,A -85,B 0,C 180,E1 -3526.334,E2 -3526.334} C_VEL
LIN {X 0,Y 547.041,Z 680.787,A -85,B 0,C 180,E1 -3527.091,E2 -3527.091} C_VEL
LIN {X 0,Y 547.328,Z 665.498,A -85,B 0,C 180,E1 -3527.709,E2 -3527.709} C_VEL
LIN {X 0,Y 547.591,Z 650.413,A -85,B 0,C 180,E1 -3528.153,E2 -3528.153} C_VEL
LIN {X 0,Y 547.801,Z 635.54,A -85,B 0,C 180,E1 -3528.443,E2 -3528.443} C_VEL
LIN {X 0,Y 548.471,Z 482.208,A -85,B 0,C 180,E1 -3530.508,E2 -3530.508} C_VEL
LIN {X 0,Y 547.031,Z 473.204,A -85,B 0,C 180,E1 -3530.711,E2 -3530.711} C_VEL
LIN {X 0,Y 547.622,Z 442.106,A -85,B 0,C 180,E1 -3533.745,E2 -3533.745} C_VEL
LIN {X 0,Y 548.205,Z 412.44,A -85,B 0,C 180,E1 -3536.661,E2 -3536.661} C_VEL
LIN {X 0,Y 548.766,Z 382.925,A -85,B 0,C 180,E1 -3539.589,E2 -3539.589} C_VEL
LIN {X 0,Y 548.854,Z 377.578,A -85,B 0,C 180,E1 -3540.124,E2 -3540.124} C_VEL
LIN {X 0,Y 545.066,Z 363.437,A -85,B 0,C 180,E1 -3541.779,E2 -3541.779} C_VEL
LIN {X 0,Y 544.986,Z 363.216,A -85,B 0,C 180,E1 -3544.571,E2 -3544.571} C_VEL
LIN {X 0,Y 544.995,Z 363.226,A -85,B 0,C 180,E1 -3547.308,E2 -3547.308} C_VEL
LIN {X 0,Y 545.006,Z 363.218,A -85,B 0,C 180,E1 -3550.149,E2 -3550.149} C_VEL
LIN {X 0,Y 545.012,Z 363.215,A -85,B 0,C 180,E1 -3552.691,E2 -3552.691} C_VEL
LIN {X 0,Y 545.013,Z 363.219,A -85,B 0,C 180,E1 -3555.173,E2 -3555.173} C_VEL
LIN {X 0,Y 545.023,Z 363.216,A -85,B 0,C 180,E1 -3558.41,E2 -3558.41} C_VEL
LIN {X 0,Y 545.046,Z 363.21,A -85,B 0,C 180,E1 -3560.815,E2 -3560.815} C_VEL
LIN {X 0,Y 545.006,Z 363.217,A -85,B 0,C 180,E1 -3563.617,E2 -3563.617} C_VEL
LIN {X 0,Y 545.038,Z 363.209,A -85,B 0,C 180,E1 -3566.326,E2 -3566.326} C_VEL
LIN {X 0,Y 545.038,Z 363.22,A -85,B 0,C 180,E1 -3568.95,E2 -3568.95} C_VEL
LIN {X 0,Y 545.041,Z 363.217,A -85,B 0,C 180,E1 -3571.504,E2 -3571.504} C_VEL
LIN {X 0,Y 545.031,Z 363.215,A -85,B 0,C 180,E1 -3573.997,E2 -3573.997} C_VEL
LIN {X 0,Y 545.073,Z 363.211,A -85,B 0,C 180,E1 -3576.44,E2 -3576.44} C_VEL
LIN {X 0,Y 545.094,Z 363.214,A -85,B 0,C 180,E1 -3579.628,E2 -3579.628} C_VEL
LIN {X 0,Y 545.117,Z 363.407,A -85,B 0,C 180,E1 -3580.025,E2 -3580.025} C_VEL
LIN {X 0,Y 545.857,Z 368.834,A -85,B 0,C 180,E1 -3581.028,E2 -3581.028} C_VEL
LIN {X 0,Y 545.729,Z 376.918,A -85,B 0,C 180,E1 -3582.388,E2 -3582.388} C_VEL
LIN {X 0,Y 547.459,Z 384.905,A -85,B 0,C 180,E1 -3582.588,E2 -3582.588} C_VEL
LIN {X 0,Y 546.892,Z 513.73,A -85,B 0,C 180,E1 -3584.358,E2 -3584.358} C_VEL
LIN {X 0,Y 546.77,Z 528.178,A -85,B 0,C 180,E1 -3584.716,E2 -3584.716} C_VEL
LIN {X 0,Y 546.508,Z 542.678,A -85,B 0,C 180,E1 -3585.239,E2 -3585.239} C_VEL
LIN {X 0,Y 546.327,Z 555.346,A -85,B 0,C 180,E1 -3585.853,E2 -3585.853} C_VEL
LIN {X 0,Y 546.025,Z 567.631,A -85,B 0,C 180,E1 -3586.604,E2 -3586.604} C_VEL
LIN {X 0,Y 545.721,Z 579.985,A -85,B 0,C 180,E1 -3587.543,E2 -3587.543} C_VEL
LIN {X 0,Y 545.459,Z 590.334,A -85,B 0,C 180,E1 -3588.504,E2 -3588.504} C_VEL
LIN {X 0,Y 545.228,Z 600.091,A -85,B 0,C 180,E1 -3589.603,E2 -3589.603} C_VEL
LIN {X 0,Y 545.024,Z 608.335,A -85,B 0,C 180,E1 -3590.724,E2 -3590.724} C_VEL
LIN {X 0,Y 544.861,Z 616.2,A -85,B 0,C 180,E1 -3592.03,E2 -3592.03} C_VEL
LIN {X 0,Y 544.756,Z 622.862,A -85,B 0,C 180,E1 -3593.413,E2 -3593.413} C_VEL
LIN {X 0,Y 544.646,Z 628.092,A -85,B 0,C 180,E1 -3594.818,E2 -3594.818} C_VEL
LIN {X 0,Y 544.659,Z 632.207,A -85,B 0,C 180,E1 -3596.301,E2 -3596.301} C_VEL
LIN {X 0,Y 544.57,Z 634.921,A -85,B 0,C 180,E1 -3597.781,E2 -3597.781} C_VEL
LIN {X 0,Y 544.537,Z 636.299,A -85,B 0,C 180,E1 -3599.26,E2 -3599.26} C_VEL
LIN {X 0,Y 544.537,Z 636.355,A -85,B 0,C 180,E1 -3600.739,E2 -3600.739} C_VEL
LIN {X 0,Y 544.568,Z 635.062,A -85,B 0,C 180,E1 -3602.219,E2 -3602.219} C_VEL
LIN {X 0,Y 544.659,Z 632.416,A -85,B 0,C 180,E1 -3603.699,E2 -3603.699} C_VEL
LIN {X 0,Y 544.645,Z 628.419,A -85,B 0,C 180,E1 -3605.182,E2 -3605.182} C_VEL
LIN {X 0,Y 544.757,Z 622.959,A -85,B 0,C 180,E1 -3606.668,E2 -3606.668} C_VEL
LIN {X 0,Y 544.854,Z 617.75,A -85,B 0,C 180,E1 -3607.784,E2 -3607.784} C_VEL
LIN {X 0,Y 545.001,Z 610.306,A -85,B 0,C 180,E1 -3609.089,E2 -3609.089} C_VEL
LIN {X 0,Y 545.165,Z 602.483,A -85,B 0,C 180,E1 -3610.21,E2 -3610.21} C_VEL
LIN {X 0,Y 545.481,Z 593.117,A -85,B 0,C 180,E1 -3611.318,E2 -3611.318} C_VEL
LIN {X 0,Y 545.708,Z 582.421,A -85,B 0,C 180,E1 -3612.363,E2 -3612.363} C_VEL
LIN {X 0,Y 546.024,Z 570.618,A -85,B 0,C 180,E1 -3613.301,E2 -3613.301} C_VEL
LIN {X 0,Y 546.264,Z 558.98,A -85,B 0,C 180,E1 -3614.054,E2 -3614.054} C_VEL
LIN {X 0,Y 546.481,Z 546.213,A -85,B 0,C 180,E1 -3614.714,E2 -3614.714} C_VEL
LIN {X 0,Y 546.707,Z 532.393,A -85,B 0,C 180,E1 -3615.255,E2 -3615.255} C_VEL
LIN {X 0,Y 546.863,Z 518.275,A -85,B 0,C 180,E1 -3615.642,E2 -3615.642} C_VEL
LIN {X 0,Y 546.95,Z 501.671,A -85,B 0,C 180,E1 -3615.918,E2 -3615.918} C_VEL
LIN {X 0,Y 547.653,Z 385.419,A -85,B 0,C 180,E1 -3617.539,E2 -3617.539} C_VEL
LIN {X 0,Y 546.149,Z 378.633,A -85,B 0,C 180,E1 -3617.719,E2 -3617.719} C_VEL
LIN {X 0,Y 546.306,Z 372.694,A -85,B 0,C 180,E1 -3618.761,E2 -3618.761} C_VEL
LIN {X 0,Y 546.171,Z 368.421,A -85,B 0,C 180,E1 -3619.546,E2 -3619.546} C_VEL
LIN {X 0,Y 545.096,Z 363.266,A -85,B 0,C 180,E1 -3620.594,E2 -3620.594} C_VEL
LIN {X 0,Y 545.058,Z 363.214,A -85,B 0,C 180,E1 -3623.725,E2 -3623.725} C_VEL
LIN {X 0,Y 545.084,Z 363.211,A -85,B 0,C 180,E1 -3626,E2 -3626} C_VEL
LIN {X 0,Y 545.094,Z 363.215,A -85,B 0,C 180,E1 -3628.748,E2 -3628.748} C_VEL
LIN {X 0,Y 545.062,Z 363.212,A -85,B 0,C 180,E1 -3631.678,E2 -3631.678} C_VEL
LIN {X 0,Y 545.066,Z 363.218,A -85,B 0,C 180,E1 -3634.564,E2 -3634.564} C_VEL
LIN {X 0,Y 545.034,Z 363.215,A -85,B 0,C 180,E1 -3637.304,E2 -3637.304} C_VEL
LIN {X 0,Y 545.068,Z 363.216,A -85,B 0,C 180,E1 -3640.142,E2 -3640.142} C_VEL
LIN {X 0,Y 545.042,Z 363.217,A -85,B 0,C 180,E1 -3642.693,E2 -3642.693} C_VEL
LIN {X 0,Y 545.024,Z 363.216,A -85,B 0,C 180,E1 -3645.171,E2 -3645.171} C_VEL
LIN {X 0,Y 545.054,Z 363.218,A -85,B 0,C 180,E1 -3647.894,E2 -3647.894} C_VEL
LIN {X 0,Y 545.078,Z 363.211,A -85,B 0,C 180,E1 -3650.817,E2 -3650.817} C_VEL
LIN {X 0,Y 545.005,Z 363.223,A -85,B 0,C 180,E1 -3653.616,E2 -3653.616} C_VEL
LIN {X 0,Y 545.037,Z 363.221,A -85,B 0,C 180,E1 -3656.325,E2 -3656.325} C_VEL
LIN {X 0,Y 545.08,Z 363.367,A -85,B 0,C 180,E1 -3659.317,E2 -3659.317} C_VEL
LIN {X 0,Y 545.717,Z 365.906,A -85,B 0,C 180,E1 -3659.639,E2 -3659.639} C_VEL
LIN {X 0,Y 548.595,Z 376.35,A -85,B 0,C 180,E1 -3660.757,E2 -3660.757} C_VEL
LIN {X 0,Y 548.193,Z 404.676,A -85,B 0,C 180,E1 -3663.338,E2 -3663.338} C_VEL
LIN {X 0,Y 547.678,Z 436.296,A -85,B 0,C 180,E1 -3666.157,E2 -3666.157} C_VEL
LIN {X 0,Y 547.168,Z 467.865,A -85,B 0,C 180,E1 -3668.921,E2 -3668.921} C_VEL
LIN {X 0,Y 547.17,Z 472.976,A -85,B 0,C 180,E1 -3669.349,E2 -3669.349} C_VEL
LIN {X 0,Y 548.508,Z 482.599,A -85,B 0,C 180,E1 -3669.544,E2 -3669.544} C_VEL
LIN {X 0,Y 547.721,Z 641.137,A -85,B 0,C 180,E1 -3671.692,E2 -3671.692} C_VEL
LIN {X 0,Y 547.552,Z 656.685,A -85,B 0,C 180,E1 -3672.057,E2 -3672.057} C_VEL
LIN {X 0,Y 547.217,Z 672.02,A -85,B 0,C 180,E1 -3672.577,E2 -3672.577} C_VEL
LIN {X 0,Y 546.95,Z 685.753,A -85,B 0,C 180,E1 -3673.194,E2 -3673.194} C_VEL
LIN {X 0,Y 546.531,Z 699.235,A -85,B 0,C 180,E1 -3673.949,E2 -3673.949} C_VEL
LIN {X 0,Y 546.154,Z 713.121,A -85,B 0,C 180,E1 -3674.907,E2 -3674.907} C_VEL
LIN {X 0,Y 545.821,Z 725.347,A -85,B 0,C 180,E1 -3675.933,E2 -3675.933} C_VEL
LIN {X 0,Y 545.512,Z 737.499,A -85,B 0,C 180,E1 -3677.159,E2 -3677.159} C_VEL
LIN {X 0,Y 545.176,Z 748.097,A -85,B 0,C 180,E1 -3678.445,E2 -3678.445} C_VEL
LIN {X 0,Y 545.051,Z 757.286,A -85,B 0,C 180,E1 -3679.787,E2 -3679.787} C_VEL
LIN {X 0,Y 544.846,Z 764.74,A -85,B 0,C 180,E1 -3681.094,E2 -3681.094} C_VEL
LIN {X 0,Y 544.746,Z 771.697,A -85,B 0,C 180,E1 -3682.586,E2 -3682.586} C_VEL
LIN {X 0,Y 544.702,Z 777.161,A -85,B 0,C 180,E1 -3684.074,E2 -3684.074} C_VEL
LIN {X 0,Y 544.606,Z 781.287,A -85,B 0,C 180,E1 -3685.558,E2 -3685.558} C_VEL
LIN {X 0,Y 544.644,Z 784.18,A -85,B 0,C 180,E1 -3687.04,E2 -3687.04} C_VEL
LIN {X 0,Y 544.543,Z 785.908,A -85,B 0,C 180,E1 -3688.52,E2 -3688.52} C_VEL
LIN {X 0,Y 544.538,Z 786.5,A -85,B 0,C 180,E1 -3689.999,E2 -3689.999} C_VEL
LIN {X 0,Y 544.543,Z 785.911,A -85,B 0,C 180,E1 -3691.478,E2 -3691.478} C_VEL
LIN {X 0,Y 544.644,Z 784.187,A -85,B 0,C 180,E1 -3692.957,E2 -3692.957} C_VEL
LIN {X 0,Y 544.605,Z 781.294,A -85,B 0,C 180,E1 -3694.44,E2 -3694.44} C_VEL
LIN {X 0,Y 544.705,Z 777.166,A -85,B 0,C 180,E1 -3695.923,E2 -3695.923} C_VEL
LIN {X 0,Y 544.744,Z 771.705,A -85,B 0,C 180,E1 -3697.411,E2 -3697.411} C_VEL
LIN {X 0,Y 544.845,Z 764.756,A -85,B 0,C 180,E1 -3698.903,E2 -3698.903} C_VEL
LIN {X 0,Y 545.073,Z 756.094,A -85,B 0,C 180,E1 -3700.398,E2 -3700.398} C_VEL
LIN {X 0,Y 545.234,Z 746.716,A -85,B 0,C 180,E1 -3701.733,E2 -3701.733} C_VEL
LIN {X 0,Y 545.509,Z 737.521,A -85,B 0,C 180,E1 -3702.839,E2 -3702.839} C_VEL
LIN {X 0,Y 545.825,Z 725.368,A -85,B 0,C 180,E1 -3704.064,E2 -3704.064} C_VEL
LIN {X 0,Y 546.189,Z 712.814,A -85,B 0,C 180,E1 -3705.114,E2 -3705.114} C_VEL
LIN {X 0,Y 546.526,Z 699.274,A -85,B 0,C 180,E1 -3706.049,E2 -3706.049} C_VEL
LIN {X 0,Y 546.941,Z 685.807,A -85,B 0,C 180,E1 -3706.804,E2 -3706.804} C_VEL
LIN {X 0,Y 547.252,Z 672.068,A -85,B 0,C 180,E1 -3707.419,E2 -3707.419} C_VEL
LIN {X 0,Y 547.545,Z 656.749,A -85,B 0,C 180,E1 -3707.94,E2 -3707.94} C_VEL
LIN {X 0,Y 547.734,Z 640.887,A -85,B 0,C 180,E1 -3708.312,E2 -3708.312} C_VEL
LIN {X 0,Y 548.499,Z 481.697,A -85,B 0,C 180,E1 -3710.469,E2 -3710.469} C_VEL
LIN {X 0,Y 547.139,Z 472.505,A -85,B 0,C 180,E1 -3710.676,E2 -3710.676} C_VEL
LIN {X 0,Y 547.682,Z 440.173,A -85,B 0,C 180,E1 -3713.539,E2 -3713.539} C_VEL
LIN {X 0,Y 548.321,Z 409.106,A -85,B 0,C 180,E1 -3716.35,E2 -3716.35} C_VEL
LIN {X 0,Y 548.973,Z 378.332,A -85,B 0,C 180,E1 -3719.198,E2 -3719.198} C_VEL
LIN {X 0,Y 548.679,Z 376.137,A -85,B 0,C 180,E1 -3719.424,E2 -3719.424} C_VEL
LIN {X 0,Y 545.097,Z 363.417,A -85,B 0,C 180,E1 -3720.877,E2 -3720.877} C_VEL
LIN {X 0,Y 545.051,Z 363.217,A -85,B 0,C 180,E1 -3722.788,E2 -3722.788} C_VEL
LIN {X 0,Y 545.007,Z 363.22,A -85,B 0,C 180,E1 -3725.669,E2 -3725.669} C_VEL
LIN {X 0,Y 545.033,Z 363.222,A -85,B 0,C 180,E1 -3728.237,E2 -3728.237} C_VEL
LIN {X 0,Y 545.008,Z 363.218,A -85,B 0,C 180,E1 -3731.119,E2 -3731.119} C_VEL
LIN {X 0,Y 545.025,Z 363.221,A -85,B 0,C 180,E1 -3734.13,E2 -3734.13} C_VEL
LIN {X 0,Y 544.985,Z 363.213,A -85,B 0,C 180,E1 -3736.884,E2 -3736.884} C_VEL
LIN {X 0,Y 545.043,Z 363.211,A -85,B 0,C 180,E1 -3739.855,E2 -3739.855} C_VEL
LIN {X 0,Y 544.996,Z 363.217,A -85,B 0,C 180,E1 -3742.693,E2 -3742.693} C_VEL
LIN {X 0,Y 545.039,Z 363.203,A -85,B 0,C 180,E1 -3745.61,E2 -3745.61} C_VEL
LIN {X 0,Y 545.042,Z 363.219,A -85,B 0,C 180,E1 -3748.321,E2 -3748.321} C_VEL
LIN {X 0,Y 545.028,Z 363.212,A -85,B 0,C 180,E1 -3751.26,E2 -3751.26} C_VEL
LIN {X 0,Y 545.036,Z 363.216,A -85,B 0,C 180,E1 -3753.997,E2 -3753.997} C_VEL
LIN {X 0,Y 545.011,Z 363.216,A -85,B 0,C 180,E1 -3757.241,E2 -3757.241} C_VEL
LIN {X 0,Y 545.085,Z 363.211,A -85,B 0,C 180,E1 -3760.414,E2 -3760.414} C_VEL
LIN {X 0,Y 545,Z 363.217,A -85,B 0,C 180,E1 -3763.519,E2 -3763.519} C_VEL
LIN {X 0,Y 545.052,Z 363.208,A -85,B 0,C 180,E1 -3765.819,E2 -3765.819} C_VEL
LIN {X 0,Y 545.092,Z 363.208,A -85,B 0,C 180,E1 -3768.849,E2 -3768.849} C_VEL
LIN {X 0,Y 545.066,Z 363.208,A -85,B 0,C 180,E1 -3771.846,E2 -3771.846} C_VEL
LIN {X 0,Y 545.148,Z 363.199,A -85,B 0,C 180,E1 -3774.822,E2 -3774.822} C_VEL
LIN {X 0,Y 545.162,Z 363.197,A -85,B 0,C 180,E1 -3777.784,E2 -3777.784} C_VEL
LIN {X 0,Y 545.194,Z 363.195,A -85,B 0,C 180,E1 -3780.739,E2 -3780.739} C_VEL
LIN {X 0,Y 545.138,Z 363.204,A -85,B 0,C 180,E1 -3782.956,E2 -3782.956} C_VEL
LIN {X 0,Y 545.111,Z 363.202,A -85,B 0,C 180,E1 -3785.92,E2 -3785.92} C_VEL
LIN {X 0,Y 545.05,Z 363.212,A -85,B 0,C 180,E1 -3788.154,E2 -3788.154} C_VEL
LIN {X 0,Y 545.093,Z 363.203,A -85,B 0,C 180,E1 -3791.151,E2 -3791.151} C_VEL
LIN {X 0,Y 545.063,Z 363.211,A -85,B 0,C 180,E1 -3794.181,E2 -3794.181} C_VEL
LIN {X 0,Y 545.056,Z 363.209,A -85,B 0,C 180,E1 -3797.421,E2 -3797.421} C_VEL
LIN {X 0,Y 545.074,Z 363.212,A -85,B 0,C 180,E1 -3800.373,E2 -3800.373} C_VEL
LIN {X 0,Y 545.055,Z 363.211,A -85,B 0,C 180,E1 -3803.561,E2 -3803.561} C_VEL
LIN {X 0,Y 545.025,Z 363.222,A -85,B 0,C 180,E1 -3806.828,E2 -3806.828} C_VEL
LIN {X 0,Y 545.007,Z 363.217,A -85,B 0,C 180,E1 -3809.342,E2 -3809.342} C_VEL
LIN {X 0,Y 545.029,Z 363.214,A -85,B 0,C 180,E1 -3811.917,E2 -3811.917} C_VEL
LIN {X 0,Y 545.042,Z 363.22,A -85,B 0,C 180,E1 -3814.566,E2 -3814.566} C_VEL
LIN {X 0,Y 545.017,Z 363.212,A -85,B 0,C 180,E1 -3817.02,E2 -3817.02} C_VEL
LIN {X 0,Y 544.337,Z 363.295,A -85,B 0,C 180,E1 -3817.637,E2 -3817.637} C_VEL
LIN {X 0,Y 541.479,Z 363.656,A -85,B 0,C 180,E1 -3818.638,E2 -3818.638} C_VEL
LIN {X 0,Y 539.075,Z 363.957,A -85,B 0,C 180,E1 -3819.444,E2 -3819.444} C_VEL
LIN {X 0,Y 538.05,Z 364.085,A -85,B 0,C 180,E1 -3820.066,E2 -3820.066} C_VEL
LIN {X 0,Y 537.969,Z 364.095,A -85,B 0,C 180,E1 -3820.277,E2 -3820.277} C_VEL
LIN {X 0,Y 537.957,Z 364.096,A -85,B 0,C 180,E1 -3822.982,E2 -3822.982} C_VEL
LIN {X 0,Y 537.985,Z 364.091,A -85,B 0,C 180,E1 -3825.931,E2 -3825.931} C_VEL
LIN {X 0,Y 537.983,Z 364.093,A -85,B 0,C 180,E1 -3829.261,E2 -3829.261} C_VEL
LIN {X 0,Y 537.972,Z 364.096,A -85,B 0,C 180,E1 -3832.123,E2 -3832.123} C_VEL
LIN {X 0,Y 537.985,Z 364.085,A -85,B 0,C 180,E1 -3835.387,E2 -3835.387} C_VEL
LIN {X 0,Y 538.006,Z 364.196,A -85,B 0,C 180,E1 -3837.973,E2 -3837.973} C_VEL
LIN {X 0,Y 538.45,Z 365.882,A -85,B 0,C 180,E1 -3838.218,E2 -3838.218} C_VEL
LIN {X 0,Y 542.061,Z 378.819,A -85,B 0,C 180,E1 -3839.732,E2 -3839.732} C_VEL
LIN {X 0,Y 541.699,Z 401.825,A -85,B 0,C 180,E1 -3842.056,E2 -3842.056} C_VEL
LIN {X 0,Y 541.128,Z 427.549,A -85,B 0,C 180,E1 -3844.623,E2 -3844.623} C_VEL
LIN {X 0,Y 540.519,Z 457.025,A -85,B 0,C 180,E1 -3847.536,E2 -3847.536} C_VEL
LIN {X 0,Y 540.204,Z 473.383,A -85,B 0,C 180,E1 -3849.122,E2 -3849.122} C_VEL
LIN {X 0,Y 541.87,Z 484.224,A -85,B 0,C 180,E1 -3849.351,E2 -3849.351} C_VEL
LIN {X 0,Y 541.001,Z 640.844,A -85,B 0,C 180,E1 -3851.5,E2 -3851.5} C_VEL
LIN {X 0,Y 540.765,Z 655.926,A -85,B 0,C 180,E1 -3851.851,E2 -3851.851} C_VEL
LIN {X 0,Y 540.481,Z 670.869,A -85,B 0,C 180,E1 -3852.355,E2 -3852.355} C_VEL
LIN {X 0,Y 540.085,Z 684.851,A -85,B 0,C 180,E1 -3852.977,E2 -3852.977} C_VEL
LIN {X 0,Y 539.671,Z 698.52,A -85,B 0,C 180,E1 -3853.742,E2 -3853.742} C_VEL
LIN {X 0,Y 539.321,Z 711.648,A -85,B 0,C 180,E1 -3854.647,E2 -3854.647} C_VEL
LIN {X 0,Y 538.939,Z 723.809,A -85,B 0,C 180,E1 -3855.656,E2 -3855.656} C_VEL
LIN {X 0,Y 538.614,Z 735.343,A -85,B 0,C 180,E1 -3856.802,E2 -3856.802} C_VEL
LIN {X 0,Y 538.259,Z 746.15,A -85,B 0,C 180,E1 -3858.085,E2 -3858.085} C_VEL
LIN {X 0,Y 538.03,Z 755.797,A -85,B 0,C 180,E1 -3859.464,E2 -3859.464} C_VEL
LIN {X 0,Y 537.841,Z 762.516,A -85,B 0,C 180,E1 -3860.601,E2 -3860.601} C_VEL
LIN {X 0,Y 537.7,Z 769.916,A -85,B 0,C 180,E1 -3862.113,E2 -3862.113} C_VEL
LIN {X 0,Y 537.596,Z 775.348,A -85,B 0,C 180,E1 -3863.489,E2 -3863.489} C_VEL
LIN {X 0,Y 537.573,Z 779.262,A -85,B 0,C 180,E1 -3864.75,E2 -3864.75} C_VEL
LIN {X 0,Y 537.561,Z 782.8,A -85,B 0,C 180,E1 -3866.253,E2 -3866.253} C_VEL
LIN {X 0,Y 537.487,Z 785.143,A -85,B 0,C 180,E1 -3867.753,E2 -3867.753} C_VEL
LIN {X 0,Y 537.437,Z 786.338,A -85,B 0,C 180,E1 -3869.252,E2 -3869.252} C_VEL
LIN {X 0,Y 537.439,Z 786.359,A -85,B 0,C 180,E1 -3870.75,E2 -3870.75} C_VEL
LIN {X 0,Y 537.488,Z 785.238,A -85,B 0,C 180,E1 -3872.249,E2 -3872.249} C_VEL
LIN {X 0,Y 537.563,Z 782.971,A -85,B 0,C 180,E1 -3873.749,E2 -3873.749} C_VEL
LIN {X 0,Y 537.573,Z 779.506,A -85,B 0,C 180,E1 -3875.252,E2 -3875.252} C_VEL
LIN {X 0,Y 537.62,Z 774.763,A -85,B 0,C 180,E1 -3876.758,E2 -3876.758} C_VEL
LIN {X 0,Y 537.728,Z 768.619,A -85,B 0,C 180,E1 -3878.267,E2 -3878.267} C_VEL
LIN {X 0,Y 537.858,Z 760.891,A -85,B 0,C 180,E1 -3879.781,E2 -3879.781} C_VEL
LIN {X 0,Y 538.082,Z 752.651,A -85,B 0,C 180,E1 -3881.109,E2 -3881.109} C_VEL
LIN {X 0,Y 538.348,Z 742.729,A -85,B 0,C 180,E1 -3882.44,E2 -3882.44} C_VEL
LIN {X 0,Y 538.66,Z 732.609,A -85,B 0,C 180,E1 -3883.584,E2 -3883.584} C_VEL
LIN {X 0,Y 539.01,Z 720.499,A -85,B 0,C 180,E1 -3884.73,E2 -3884.73} C_VEL
LIN {X 0,Y 539.458,Z 708.514,A -85,B 0,C 180,E1 -3885.678,E2 -3885.678} C_VEL
LIN {X 0,Y 539.841,Z 695.288,A -85,B 0,C 180,E1 -3886.547,E2 -3886.547} C_VEL
LIN {X 0,Y 540.211,Z 680.766,A -85,B 0,C 180,E1 -3887.314,E2 -3887.314} C_VEL
LIN {X 0,Y 540.56,Z 665.469,A -85,B 0,C 180,E1 -3887.938,E2 -3887.938} C_VEL
LIN {X 0,Y 540.861,Z 650.24,A -85,B 0,C 180,E1 -3888.39,E2 -3888.39} C_VEL
LIN {X 0,Y 541.071,Z 634.746,A -85,B 0,C 180,E1 -3888.692,E2 -3888.692} C_VEL
LIN {X 0,Y 541.799,Z 482.892,A -85,B 0,C 180,E1 -3890.76,E2 -3890.76} C_VEL
LIN {X 0,Y 540.211,Z 473.311,A -85,B 0,C 180,E1 -3890.971,E2 -3890.971} C_VEL
LIN {X 0,Y 540.797,Z 442.869,A -85,B 0,C 180,E1 -3893.954,E2 -3893.954} C_VEL
LIN {X 0,Y 541.399,Z 415.842,A -85,B 0,C 180,E1 -3896.632,E2 -3896.632} C_VEL
LIN {X 0,Y 542.017,Z 387.066,A -85,B 0,C 180,E1 -3899.521,E2 -3899.521} C_VEL
LIN {X 0,Y 542.006,Z 378.667,A -85,B 0,C 180,E1 -3900.379,E2 -3900.379} C_VEL
LIN {X 0,Y 538.012,Z 364.311,A -85,B 0,C 180,E1 -3902.082,E2 -3902.082} C_VEL
LIN {X 0,Y 537.941,Z 364.09,A -85,B 0,C 180,E1 -3904.18,E2 -3904.18} C_VEL
LIN {X 0,Y 537.952,Z 364.101,A -85,B 0,C 180,E1 -3907.162,E2 -3907.162} C_VEL
LIN {X 0,Y 537.965,Z 364.097,A -85,B 0,C 180,E1 -3909.803,E2 -3909.803} C_VEL
LIN {X 0,Y 537.962,Z 364.094,A -85,B 0,C 180,E1 -3912.793,E2 -3912.793} C_VEL
LIN {X 0,Y 537.986,Z 364.094,A -85,B 0,C 180,E1 -3915.136,E2 -3915.136} C_VEL
LIN {X 0,Y 537.981,Z 364.092,A -85,B 0,C 180,E1 -3918.222,E2 -3918.222} C_VEL
LIN {X 0,Y 537.986,Z 364.095,A -85,B 0,C 180,E1 -3921.167,E2 -3921.167} C_VEL
LIN {X 0,Y 537.962,Z 364.091,A -85,B 0,C 180,E1 -3924.094,E2 -3924.094} C_VEL
LIN {X 0,Y 538.002,Z 364.088,A -85,B 0,C 180,E1 -3926.725,E2 -3926.725} C_VEL
LIN {X 0,Y 537.994,Z 364.094,A -85,B 0,C 180,E1 -3929.563,E2 -3929.563} C_VEL
LIN {X 0,Y 537.994,Z 364.094,A -85,B 0,C 180,E1 -3932.662,E2 -3932.662} C_VEL
LIN {X 0,Y 537.972,Z 364.101,A -85,B 0,C 180,E1 -3935.289,E2 -3935.289} C_VEL
LIN {X 0,Y 538.019,Z 364.091,A -85,B 0,C 180,E1 -3938.043,E2 -3938.043} C_VEL
LIN {X 0,Y 538.087,Z 364.228,A -85,B 0,C 180,E1 -3939.832,E2 -3939.832} C_VEL
LIN {X 0,Y 538.96,Z 370.408,A -85,B 0,C 180,E1 -3940.974,E2 -3940.974} C_VEL
LIN {X 0,Y 538.863,Z 377.433,A -85,B 0,C 180,E1 -3942.154,E2 -3942.154} C_VEL
LIN {X 0,Y 540.715,Z 386.748,A -85,B 0,C 180,E1 -3942.38,E2 -3942.38} C_VEL
LIN {X 0,Y 540.034,Z 514.553,A -85,B 0,C 180,E1 -3944.173,E2 -3944.173} C_VEL
LIN {X 0,Y 539.873,Z 529.257,A -85,B 0,C 180,E1 -3944.544,E2 -3944.544} C_VEL
LIN {X 0,Y 539.658,Z 543.008,A -85,B 0,C 180,E1 -3945.047,E2 -3945.047} C_VEL
LIN {X 0,Y 539.467,Z 555.785,A -85,B 0,C 180,E1 -3945.669,E2 -3945.669} C_VEL
LIN {X 0,Y 539.166,Z 566.774,A -85,B 0,C 180,E1 -3946.334,E2 -3946.334} C_VEL
LIN {X 0,Y 538.86,Z 578.33,A -85,B 0,C 180,E1 -3947.19,E2 -3947.19} C_VEL
LIN {X 0,Y 538.578,Z 588.994,A -85,B 0,C 180,E1 -3948.152,E2 -3948.152} C_VEL
LIN {X 0,Y 538.367,Z 599.273,A -85,B 0,C 180,E1 -3949.279,E2 -3949.279} C_VEL
LIN {X 0,Y 538.11,Z 607.86,A -85,B 0,C 180,E1 -3950.414,E2 -3950.414} C_VEL
LIN {X 0,Y 537.893,Z 616.029,A -85,B 0,C 180,E1 -3951.737,E2 -3951.737} C_VEL
LIN {X 0,Y 537.781,Z 621.745,A -85,B 0,C 180,E1 -3952.868,E2 -3952.868} C_VEL
LIN {X 0,Y 537.724,Z 627.737,A -85,B 0,C 180,E1 -3954.375,E2 -3954.375} C_VEL
LIN {X 0,Y 537.629,Z 631.217,A -85,B 0,C 180,E1 -3955.501,E2 -3955.501} C_VEL
LIN {X 0,Y 537.601,Z 634.545,A -85,B 0,C 180,E1 -3957.002,E2 -3957.002} C_VEL
LIN {X 0,Y 537.489,Z 636.55,A -85,B 0,C 180,E1 -3958.501,E2 -3958.501} C_VEL
LIN {X 0,Y 537.481,Z 637.266,A -85,B 0,C 180,E1 -3960,E2 -3960} C_VEL
LIN {X 0,Y 537.489,Z 636.683,A -85,B 0,C 180,E1 -3961.498,E2 -3961.498} C_VEL
LIN {X 0,Y 537.609,Z 634.784,A -85,B 0,C 180,E1 -3962.997,E2 -3962.997} C_VEL
LIN {X 0,Y 537.638,Z 631.562,A -85,B 0,C 180,E1 -3964.498,E2 -3964.498} C_VEL
LIN {X 0,Y 537.759,Z 626.898,A -85,B 0,C 180,E1 -3966.001,E2 -3966.001} C_VEL
LIN {X 0,Y 537.782,Z 622.354,A -85,B 0,C 180,E1 -3967.132,E2 -3967.132} C_VEL
LIN {X 0,Y 537.962,Z 615.753,A -85,B 0,C 180,E1 -3968.451,E2 -3968.451} C_VEL
LIN {X 0,Y 538.134,Z 607.538,A -85,B 0,C 180,E1 -3969.775,E2 -3969.775} C_VEL
LIN {X 0,Y 538.424,Z 598.885,A -85,B 0,C 180,E1 -3970.91,E2 -3970.91} C_VEL
LIN {X 0,Y 538.707,Z 588.36,A -85,B 0,C 180,E1 -3972.048,E2 -3972.048} C_VEL
LIN {X 0,Y 538.963,Z 577.658,A -85,B 0,C 180,E1 -3972.999,E2 -3972.999} C_VEL
LIN {X 0,Y 539.214,Z 565.868,A -85,B 0,C 180,E1 -3973.857,E2 -3973.857} C_VEL
LIN {X 0,Y 539.56,Z 552.743,A -85,B 0,C 180,E1 -3974.618,E2 -3974.618} C_VEL
LIN {X 0,Y 539.827,Z 540.617,A -85,B 0,C 180,E1 -3975.167,E2 -3975.167} C_VEL
LIN {X 0,Y 539.967,Z 526.562,A -85,B 0,C 180,E1 -3975.642,E2 -3975.642} C_VEL
LIN {X 0,Y 540.081,Z 512.728,A -85,B 0,C 180,E1 -3975.956,E2 -3975.956} C_VEL
LIN {X 0,Y 540.943,Z 386.692,A -85,B 0,C 180,E1 -3977.774,E2 -3977.774} C_VEL
LIN {X 0,Y 539.525,Z 380.237,A -85,B 0,C 180,E1 -3977.935,E2 -3977.935} C_VEL
LIN {X 0,Y 539.365,Z 379.037,A -85,B 0,C 180,E1 -3978.036,E2 -3978.036} C_VEL
LIN {X 0,Y 539.43,Z 370.498,A -85,B 0,C 180,E1 -3979.602,E2 -3979.602} C_VEL
LIN {X 0,Y 538.06,Z 364.143,A -85,B 0,C 180,E1 -3980.901,E2 -3980.901} C_VEL
LIN {X 0,Y 538.005,Z 364.093,A -85,B 0,C 180,E1 -3983.888,E2 -3983.888} C_VEL
LIN {X 0,Y 538.046,Z 364.091,A -85,B 0,C 180,E1 -3986.366,E2 -3986.366} C_VEL
LIN {X 0,Y 538.035,Z 364.093,A -85,B 0,C 180,E1 -3988.933,E2 -3988.933} C_VEL
LIN {X 0,Y 538.014,Z 364.091,A -85,B 0,C 180,E1 -3991.887,E2 -3991.887} C_VEL
LIN {X 0,Y 538.016,Z 364.096,A -85,B 0,C 180,E1 -3994.617,E2 -3994.617} C_VEL
LIN {X 0,Y 538.003,Z 364.092,A -85,B 0,C 180,E1 -3997.169,E2 -3997.169} C_VEL
LIN {X 0,Y 538.025,Z 364.09,A -85,B 0,C 180,E1 -3999.797,E2 -3999.797} C_VEL
LIN {X 0,Y 537.991,Z 364.095,A -85,B 0,C 180,E1 -4002.789,E2 -4002.789} C_VEL
LIN {X 0,Y 537.997,Z 364.092,A -85,B 0,C 180,E1 -4005.136,E2 -4005.136} C_VEL
LIN {X 0,Y 538,Z 364.098,A -85,B 0,C 180,E1 -4008.223,E2 -4008.223} C_VEL
LIN {X 0,Y 538.01,Z 364.091,A -85,B 0,C 180,E1 -4011.168,E2 -4011.168} C_VEL
LIN {X 0,Y 537.96,Z 364.102,A -85,B 0,C 180,E1 -4014.094,E2 -4014.094} C_VEL
LIN {X 0,Y 538.001,Z 364.095,A -85,B 0,C 180,E1 -4016.724,E2 -4016.724} C_VEL
LIN {X 0,Y 538.043,Z 364.318,A -85,B 0,C 180,E1 -4019.058,E2 -4019.058} C_VEL
LIN {X 0,Y 541.627,Z 377.601,A -85,B 0,C 180,E1 -4020.557,E2 -4020.557} C_VEL
LIN {X 0,Y 541.851,Z 382.192,A -85,B 0,C 180,E1 -4021.002,E2 -4021.002} C_VEL
LIN {X 0,Y 541.179,Z 414.84,A -85,B 0,C 180,E1 -4024.004,E2 -4024.004} C_VEL
LIN {X 0,Y 540.608,Z 447.59,A -85,B 0,C 180,E1 -4026.943,E2 -4026.943} C_VEL
LIN {X 0,Y 540.188,Z 472.123,A -85,B 0,C 180,E1 -4029.095,E2 -4029.095} C_VEL
LIN {X 0,Y 541.792,Z 483.102,A -85,B 0,C 180,E1 -4029.314,E2 -4029.314} C_VEL
LIN {X 0,Y 541.017,Z 639.869,A -85,B 0,C 180,E1 -4031.436,E2 -4031.436} C_VEL
LIN {X 0,Y 540.797,Z 655.387,A -85,B 0,C 180,E1 -4031.79,E2 -4031.79} C_VEL
LIN {X 0,Y 540.481,Z 670.786,A -85,B 0,C 180,E1 -4032.304,E2 -4032.304} C_VEL
LIN {X 0,Y 540.173,Z 683.772,A -85,B 0,C 180,E1 -4032.88,E2 -4032.88} C_VEL
LIN {X 0,Y 539.732,Z 697.653,A -85,B 0,C 180,E1 -4033.644,E2 -4033.644} C_VEL
LIN {X 0,Y 539.364,Z 710.482,A -85,B 0,C 180,E1 -4034.514,E2 -4034.514} C_VEL
LIN {X 0,Y 538.945,Z 723.215,A -85,B 0,C 180,E1 -4035.557,E2 -4035.557} C_VEL
LIN {X 0,Y 538.613,Z 733.956,A -85,B 0,C 180,E1 -4036.607,E2 -4036.607} C_VEL
LIN {X 0,Y 538.307,Z 743.895,A -85,B 0,C 180,E1 -4037.75,E2 -4037.75} C_VEL
LIN {X 0,Y 538.097,Z 753.615,A -85,B 0,C 180,E1 -4039.082,E2 -4039.082} C_VEL
LIN {X 0,Y 537.825,Z 761.714,A -85,B 0,C 180,E1 -4040.408,E2 -4040.408} C_VEL
LIN {X 0,Y 537.735,Z 768.416,A -85,B 0,C 180,E1 -4041.733,E2 -4041.733} C_VEL
LIN {X 0,Y 537.619,Z 774.605,A -85,B 0,C 180,E1 -4043.242,E2 -4043.242} C_VEL
LIN {X 0,Y 537.574,Z 779.384,A -85,B 0,C 180,E1 -4044.748,E2 -4044.748} C_VEL
LIN {X 0,Y 537.562,Z 782.882,A -85,B 0,C 180,E1 -4046.251,E2 -4046.251} C_VEL
LIN {X 0,Y 537.486,Z 785.186,A -85,B 0,C 180,E1 -4047.751,E2 -4047.751} C_VEL
LIN {X 0,Y 537.439,Z 786.347,A -85,B 0,C 180,E1 -4049.25,E2 -4049.25} C_VEL
LIN {X 0,Y 537.439,Z 786.348,A -85,B 0,C 180,E1 -4050.748,E2 -4050.748} C_VEL
LIN {X 0,Y 537.486,Z 785.191,A -85,B 0,C 180,E1 -4052.247,E2 -4052.247} C_VEL
LIN {X 0,Y 537.561,Z 782.89,A -85,B 0,C 180,E1 -4053.747,E2 -4053.747} C_VEL
LIN {X 0,Y 537.574,Z 779.389,A -85,B 0,C 180,E1 -4055.25,E2 -4055.25} C_VEL
LIN {X 0,Y 537.617,Z 774.61,A -85,B 0,C 180,E1 -4056.755,E2 -4056.755} C_VEL
LIN {X 0,Y 537.733,Z 768.429,A -85,B 0,C 180,E1 -4058.265,E2 -4058.265} C_VEL
LIN {X 0,Y 537.872,Z 760.656,A -85,B 0,C 180,E1 -4059.778,E2 -4059.778} C_VEL
LIN {X 0,Y 538.1,Z 752.376,A -85,B 0,C 180,E1 -4061.106,E2 -4061.106} C_VEL
LIN {X 0,Y 538.356,Z 742.402,A -85,B 0,C 180,E1 -4062.438,E2 -4062.438} C_VEL
LIN {X 0,Y 538.661,Z 732.197,A -85,B 0,C 180,E1 -4063.581,E2 -4063.581} C_VEL
LIN {X 0,Y 539.019,Z 720.026,A -85,B 0,C 180,E1 -4064.728,E2 -4064.728} C_VEL
LIN {X 0,Y 539.461,Z 707.84,A -85,B 0,C 180,E1 -4065.681,E2 -4065.681} C_VEL
LIN {X 0,Y 539.834,Z 694.535,A -85,B 0,C 180,E1 -4066.545,E2 -4066.545} C_VEL
LIN {X 0,Y 540.234,Z 679.851,A -85,B 0,C 180,E1 -4067.311,E2 -4067.311} C_VEL
LIN {X 0,Y 540.624,Z 664.328,A -85,B 0,C 180,E1 -4067.933,E2 -4067.933} C_VEL
LIN {X 0,Y 540.927,Z 648.538,A -85,B 0,C 180,E1 -4068.387,E2 -4068.387} C_VEL
LIN {X 0,Y 541.083,Z 633.136,A -85,B 0,C 180,E1 -4068.671,E2 -4068.671} C_VEL
LIN {X 0,Y 541.776,Z 482.269,A -85,B 0,C 180,E1 -4070.704,E2 -4070.704} C_VEL
LIN {X 0,Y 540.242,Z 472.216,A -85,B 0,C 180,E1 -4070.917,E2 -4070.917} C_VEL
LIN {X 0,Y 540.843,Z 440.555,A -85,B 0,C 180,E1 -4073.754,E2 -4073.754} C_VEL
LIN {X 0,Y 541.554,Z 410.304,A -85,B 0,C 180,E1 -4076.534,E2 -4076.534} C_VEL
LIN {X 0,Y 542.286,Z 379.733,A -85,B 0,C 180,E1 -4079.404,E2 -4079.404} C_VEL
LIN {X 0,Y 538.051,Z 364.283,A -85,B 0,C 180,E1 -4081.182,E2 -4081.182} C_VEL
LIN {X 0,Y 537.987,Z 364.098,A -85,B 0,C 180,E1 -4084.174,E2 -4084.174} C_VEL
LIN {X 0,Y 537.952,Z 364.097,A -85,B 0,C 180,E1 -4087.163,E2 -4087.163} C_VEL
LIN {X 0,Y 537.993,Z 364.094,A -85,B 0,C 180,E1 -4089.798,E2 -4089.798} C_VEL
LIN {X 0,Y 537.975,Z 364.096,A -85,B 0,C 180,E1 -4092.788,E2 -4092.788} C_VEL
LIN {X 0,Y 537.976,Z 364.093,A -85,B 0,C 180,E1 -4095.135,E2 -4095.135} C_VEL
LIN {X 0,Y 537.97,Z 364.089,A -85,B 0,C 180,E1 -4098.221,E2 -4098.221} C_VEL
LIN {X 0,Y 537.992,Z 364.091,A -85,B 0,C 180,E1 -4101.168,E2 -4101.168} C_VEL
LIN {X 0,Y 537.946,Z 364.093,A -85,B 0,C 180,E1 -4104.093,E2 -4104.093} C_VEL
LIN {X 0,Y 538.017,Z 364.09,A -85,B 0,C 180,E1 -4106.727,E2 -4106.727} C_VEL
LIN {X 0,Y 537.989,Z 364.091,A -85,B 0,C 180,E1 -4109.56,E2 -4109.56} C_VEL
LIN {X 0,Y 537.989,Z 364.097,A -85,B 0,C 180,E1 -4112.658,E2 -4112.658} C_VEL
LIN {X 0,Y 537.966,Z 364.089,A -85,B 0,C 180,E1 -4115.289,E2 -4115.289} C_VEL
LIN {X 0,Y 537.998,Z 364.093,A -85,B 0,C 180,E1 -4118.042,E2 -4118.042} C_VEL
LIN {X 0,Y 537.989,Z 364.093,A -85,B 0,C 180,E1 -4120.938,E2 -4120.938} C_VEL
LIN {X 0,Y 537.947,Z 364.096,A -85,B 0,C 180,E1 -4123.297,E2 -4123.297} C_VEL
LIN {X 0,Y 538.024,Z 364.082,A -85,B 0,C 180,E1 -4125.63,E2 -4125.63} C_VEL
LIN {X 0,Y 538.053,Z 364.087,A -85,B 0,C 180,E1 -4128.701,E2 -4128.701} C_VEL
LIN {X 0,Y 538.029,Z 364.084,A -85,B 0,C 180,E1 -4131.739,E2 -4131.739} C_VEL
LIN {X 0,Y 538.107,Z 364.077,A -85,B 0,C 180,E1 -4134.755,E2 -4134.755} C_VEL
LIN {X 0,Y 538.135,Z 364.072,A -85,B 0,C 180,E1 -4137.755,E2 -4137.755} C_VEL
LIN {X 0,Y 538.164,Z 364.071,A -85,B 0,C 180,E1 -4140.748,E2 -4140.748} C_VEL
LIN {X 0,Y 538.104,Z 364.08,A -85,B 0,C 180,E1 -4142.995,E2 -4142.995} C_VEL
LIN {X 0,Y 538.068,Z 364.08,A -85,B 0,C 180,E1 -4145.998,E2 -4145.998} C_VEL
LIN {X 0,Y 538.021,Z 364.088,A -85,B 0,C 180,E1 -4148.261,E2 -4148.261} C_VEL
LIN {X 0,Y 538.066,Z 364.076,A -85,B 0,C 180,E1 -4151.597,E2 -4151.597} C_VEL
LIN {X 0,Y 538.032,Z 364.089,A -85,B 0,C 180,E1 -4154.853,E2 -4154.853} C_VEL
LIN {X 0,Y 538.02,Z 364.085,A -85,B 0,C 180,E1 -4157.533,E2 -4157.533} C_VEL
LIN {X 0,Y 538.02,Z 364.092,A -85,B 0,C 180,E1 -4160.652,E2 -4160.652} C_VEL
LIN {X 0,Y 537.991,Z 364.091,A -85,B 0,C 180,E1 -4163.878,E2 -4163.878} C_VEL
LIN {X 0,Y 537.962,Z 364.096,A -85,B 0,C 180,E1 -4166.371,E2 -4166.371} C_VEL
LIN {X 0,Y 537.977,Z 364.097,A -85,B 0,C 180,E1 -4168.927,E2 -4168.927} C_VEL
LIN {X 0,Y 537.984,Z 364.092,A -85,B 0,C 180,E1 -4171.886,E2 -4171.886} C_VEL
LIN {X 0,Y 537.992,Z 364.099,A -85,B 0,C 180,E1 -4174.618,E2 -4174.618} C_VEL
LIN {X 0,Y 537.971,Z 364.088,A -85,B 0,C 180,E1 -4177.168,E2 -4177.168} C_VEL
